KUKA KRL program: EPS_2_25748_MH02A_A_20260121065856.src

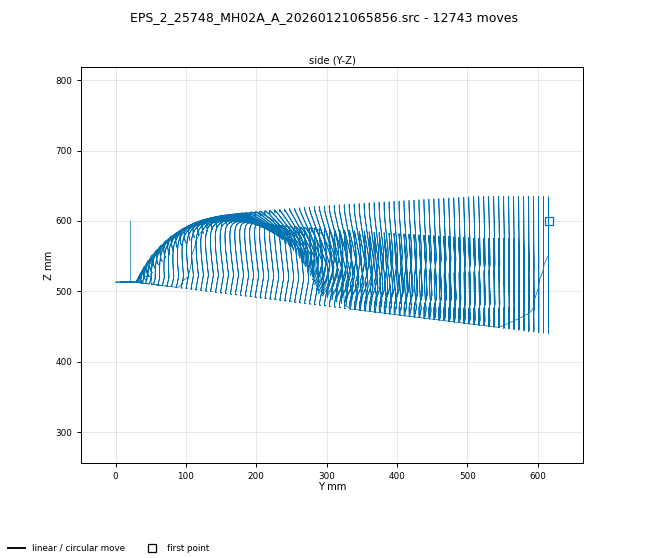
[picture p0: tool path of EPS_2_25748_MH02A_A_20260121065856.src, 12743 of 12745 moves have a stored position in this frame; points joined in program order, loops and branches not executed]
&ACCESS RVP
&REL 4
&COMMENT QRS 19112012
&PARAM EDITMASK = *
DEF PART()
EXT BAS (BAS_COMMAND :IN,REAL :IN )
INT I
BAS (#INITMOV,0 )

;KUKA QRS Post kuka4.cps  Date:22-06-2017 !

File_ID=2997

QRS_PRE_INIT()

;Init var - Until changes are made in qrs_pre_init
Outlet_Square_prg=0
Inlet_1_Square_prg=0
Inlet_2_Square_prg=0
Inlet_3_Square_prg=0
Inlet_4_Square_prg=0
Inlet_5_Square_prg=0

Outlet_1={X 0.000, Y 515.340, Z 534.500, B 0.000, E1 0.000 }
Inlet_1={X 0.000, Y 519.690, Z 474.500, B 0.000, E1 90.000 }
Inlet_2={X 0.000, Y 519.690, Z 474.500, B 0.000, E1 270.000 }
Outlet_1_type=201
Inlet_1_type=201
Inlet_2_type=201
;QRS#1=Sidecore dimensions
;QRS#2=200-8" PVC SDR 35
;QRS#3=200-8" PVC SDR 35
;QRS#4=200-8" PVC SDR 35
;QRS#5=
;QRS#6=
;QRS#7=
;QRS#8=
;QRS#9=12-08 PSX
;QRS#10=12-08 PSX
;QRS#11=12-08 PSX
;QRS#12=
;QRS#13=
;QRS#14=
;QRS#15=
;QRS#16=1220x127x914 3'
;QRS#17=EPS Height
;QRS#18=635
;QRS#19=*
;QRS#20= UPDATED VERSION 22-06-2017
;QRS#21=*
Outlet_Square=0100
Inlet_1_Square=0100
Inlet_2_Square=0100
Inlet_3_Square=0
Inlet_4_Square=0
Inlet_5_Square=0
Mill_Square=1
Outlet_Square_Prg=204
Inlet_1_Square_prg=204
Inlet_2_Square_prg=204

QRS_INIT()

$ADVANCE=5

; T1
PTP {E1 173.497,E2 173.497}
PTP {X 0,Y 615.499,A -85,B 0,C 180,E1 173.497,E2 173.497,E3 0,E4 0,E5 0,E6 0}
QRS_SPEED_INIT()
LIN {X 0,Y 615.499,Z 600,A -85,B 0,C 180,E1 173.497,E2 173.497,E3 0,E4 0,E5 0,E6 0} C_VEL
LIN {X 0,Y 615.499,Z 565.725,A -85,B 0,C 180,E1 173.497,E2 173.497} C_VEL
LIN {X 0,Y 615.499,Z 554.844,A -85,B 0,C 180,E1 173.497,E2 173.497} C_VEL
LIN {X 0,Y 615.497,Z 553.2,A -85,B 0,C 180,E1 173.417,E2 173.417} C_VEL
LIN {X 0,Y 615.497,Z 545.535,A -85,B 0,C 180,E1 172.454,E2 172.454} C_VEL
LIN {X 0,Y 615.498,Z 535.756,A -85,B 0,C 180,E1 171.463,E2 171.463} C_VEL
LIN {X 0,Y 615.498,Z 525.49,A -85,B 0,C 180,E1 170.635,E2 170.635} C_VEL
LIN {X 0,Y 615.481,Z 513.928,A -85,B 0,C 180,E1 169.888,E2 169.888} C_VEL
LIN {X 0,Y 615.482,Z 502.142,A -85,B 0,C 180,E1 169.296,E2 169.296} C_VEL
LIN {X 0,Y 615.483,Z 489.153,A -85,B 0,C 180,E1 168.807,E2 168.807} C_VEL
LIN {X 0,Y 615.487,Z 476.549,A -85,B 0,C 180,E1 168.473,E2 168.473} C_VEL
LIN {X 0,Y 615.484,Z 471.197,A -85,B 0,C 180,E1 168.369,E2 168.369} C_VEL
LIN {X 0,Y 615.476,Z 467.928,A -85,B 0,C 180,E1 166.073,E2 166.073} C_VEL
LIN {X 0,Y 615.492,Z 464.179,A -85,B 0,C 180,E1 163.413,E2 163.413} C_VEL
LIN {X 0,Y 615.485,Z 460.37,A -85,B 0,C 180,E1 160.662,E2 160.662} C_VEL
LIN {X 0,Y 615.48,Z 456.547,A -85,B 0,C 180,E1 157.863,E2 157.863} C_VEL
LIN {X 0,Y 615.476,Z 452.731,A -85,B 0,C 180,E1 155.007,E2 155.007} C_VEL
LIN {X 0,Y 615.481,Z 449.861,A -85,B 0,C 180,E1 152.822,E2 152.822} C_VEL
LIN {X 0,Y 615.498,Z 446.504,A -85,B 0,C 180,E1 150.204,E2 150.204} C_VEL
LIN {X 0,Y 615.485,Z 443.191,A -85,B 0,C 180,E1 147.542,E2 147.542} C_VEL
LIN {X 0,Y 615.48,Z 440.363,A -85,B 0,C 180,E1 145.184,E2 145.184} C_VEL
LIN {X 0,Y 615.477,Z 439.691,A -85,B 0,C 180,E1 144.168,E2 144.168} C_VEL
LIN {X 0,Y 615.484,Z 439.689,A -85,B 0,C 180,E1 141.931,E2 141.931} C_VEL
LIN {X 0,Y 615.479,Z 439.698,A -85,B 0,C 180,E1 139.392,E2 139.392} C_VEL
LIN {X 0,Y 615.497,Z 439.687,A -85,B 0,C 180,E1 136.756,E2 136.756} C_VEL
LIN {X 0,Y 615.49,Z 439.69,A -85,B 0,C 180,E1 133.997,E2 133.997} C_VEL
LIN {X 0,Y 615.491,Z 439.7,A -85,B 0,C 180,E1 131.094,E2 131.094} C_VEL
LIN {X 0,Y 615.486,Z 439.692,A -85,B 0,C 180,E1 128.905,E2 128.905} C_VEL
LIN {X 0,Y 615.479,Z 439.691,A -85,B 0,C 180,E1 126.426,E2 126.426} C_VEL
LIN {X 0,Y 615.496,Z 439.697,A -85,B 0,C 180,E1 124.022,E2 124.022} C_VEL
LIN {X 0,Y 615.487,Z 439.688,A -85,B 0,C 180,E1 121.686,E2 121.686} C_VEL
LIN {X 0,Y 615.484,Z 439.693,A -85,B 0,C 180,E1 119.407,E2 119.407} C_VEL
LIN {X 0,Y 615.486,Z 439.696,A -85,B 0,C 180,E1 117.044,E2 117.044} C_VEL
LIN {X 0,Y 615.477,Z 439.694,A -85,B 0,C 180,E1 114.273,E2 114.273} C_VEL
LIN {X 0,Y 615.477,Z 439.69,A -85,B 0,C 180,E1 111.432,E2 111.432} C_VEL
LIN {X 0,Y 615.491,Z 439.699,A -85,B 0,C 180,E1 108.604,E2 108.604} C_VEL
LIN {X 0,Y 615.489,Z 439.688,A -85,B 0,C 180,E1 105.905,E2 105.905} C_VEL
LIN {X 0,Y 615.482,Z 439.694,A -85,B 0,C 180,E1 103.201,E2 103.201} C_VEL
LIN {X 0,Y 615.478,Z 439.694,A -85,B 0,C 180,E1 100.527,E2 100.527} C_VEL
LIN {X 0,Y 615.489,Z 439.689,A -85,B 0,C 180,E1 97.876,E2 97.876} C_VEL
LIN {X 0,Y 615.482,Z 439.696,A -85,B 0,C 180,E1 95.241,E2 95.241} C_VEL
LIN {X 0,Y 615.477,Z 439.691,A -85,B 0,C 180,E1 92.618,E2 92.618} C_VEL
LIN {X 0,Y 615.492,Z 439.696,A -85,B 0,C 180,E1 90,E2 90} C_VEL
LIN {X 0,Y 615.478,Z 439.69,A -85,B 0,C 180,E1 87.382,E2 87.382} C_VEL
LIN {X 0,Y 615.494,Z 439.698,A -85,B 0,C 180,E1 84.759,E2 84.759} C_VEL
LIN {X 0,Y 615.487,Z 439.688,A -85,B 0,C 180,E1 82.124,E2 82.124} C_VEL
LIN {X 0,Y 615.494,Z 439.7,A -85,B 0,C 180,E1 79.473,E2 79.473} C_VEL
LIN {X 0,Y 615.482,Z 439.689,A -85,B 0,C 180,E1 76.799,E2 76.799} C_VEL
LIN {X 0,Y 615.491,Z 439.694,A -85,B 0,C 180,E1 74.095,E2 74.095} C_VEL
LIN {X 0,Y 615.483,Z 439.693,A -85,B 0,C 180,E1 71.354,E2 71.354} C_VEL
LIN {X 0,Y 615.477,Z 439.691,A -85,B 0,C 180,E1 68.568,E2 68.568} C_VEL
LIN {X 0,Y 615.485,Z 439.701,A -85,B 0,C 180,E1 65.728,E2 65.728} C_VEL
LIN {X 0,Y 615.486,Z 439.689,A -85,B 0,C 180,E1 62.956,E2 62.956} C_VEL
LIN {X 0,Y 615.498,Z 439.689,A -85,B 0,C 180,E1 60.205,E2 60.205} C_VEL
LIN {X 0,Y 615.48,Z 439.695,A -85,B 0,C 180,E1 57.542,E2 57.542} C_VEL
LIN {X 0,Y 615.499,Z 439.691,A -85,B 0,C 180,E1 55.185,E2 55.185} C_VEL
LIN {X 0,Y 615.477,Z 439.69,A -85,B 0,C 180,E1 52.757,E2 52.757} C_VEL
LIN {X 0,Y 615.477,Z 439.694,A -85,B 0,C 180,E1 49.913,E2 49.913} C_VEL
LIN {X 0,Y 615.475,Z 439.69,A -85,B 0,C 180,E1 47.646,E2 47.646} C_VEL
LIN {X 0,Y 615.483,Z 439.696,A -85,B 0,C 180,E1 44.931,E2 44.931} C_VEL
LIN {X 0,Y 615.494,Z 439.692,A -85,B 0,C 180,E1 42.08,E2 42.08} C_VEL
LIN {X 0,Y 615.478,Z 439.696,A -85,B 0,C 180,E1 39.751,E2 39.751} C_VEL
LIN {X 0,Y 615.485,Z 439.694,A -85,B 0,C 180,E1 36.936,E2 36.936} C_VEL
LIN {X 0,Y 615.48,Z 439.689,A -85,B 0,C 180,E1 35.617,E2 35.617} C_VEL
LIN {X 0,Y 615.493,Z 440.123,A -85,B 0,C 180,E1 34.701,E2 34.701} C_VEL
LIN {X 0,Y 615.495,Z 443.189,A -85,B 0,C 180,E1 32.331,E2 32.331} C_VEL
LIN {X 0,Y 615.487,Z 446.882,A -85,B 0,C 180,E1 29.407,E2 29.407} C_VEL
LIN {X 0,Y 615.48,Z 449.92,A -85,B 0,C 180,E1 27.043,E2 27.043} C_VEL
LIN {X 0,Y 615.492,Z 453.568,A -85,B 0,C 180,E1 24.272,E2 24.272} C_VEL
LIN {X 0,Y 615.494,Z 457.377,A -85,B 0,C 180,E1 21.432,E2 21.432} C_VEL
LIN {X 0,Y 615.494,Z 461.252,A -85,B 0,C 180,E1 18.606,E2 18.606} C_VEL
LIN {X 0,Y 615.476,Z 465.011,A -85,B 0,C 180,E1 15.906,E2 15.906} C_VEL
LIN {X 0,Y 615.493,Z 468.827,A -85,B 0,C 180,E1 13.201,E2 13.201} C_VEL
LIN {X 0,Y 615.484,Z 471.187,A -85,B 0,C 180,E1 11.548,E2 11.548} C_VEL
LIN {X 0,Y 615.485,Z 486.247,A -85,B 0,C 180,E1 11.193,E2 11.193} C_VEL
LIN {X 0,Y 615.48,Z 497.908,A -85,B 0,C 180,E1 10.793,E2 10.793} C_VEL
LIN {X 0,Y 615.486,Z 509.192,A -85,B 0,C 180,E1 10.278,E2 10.278} C_VEL
LIN {X 0,Y 615.492,Z 520.573,A -85,B 0,C 180,E1 9.613,E2 9.613} C_VEL
LIN {X 0,Y 615.498,Z 530.82,A -85,B 0,C 180,E1 8.868,E2 8.868} C_VEL
LIN {X 0,Y 615.498,Z 540.032,A -85,B 0,C 180,E1 8.041,E2 8.041} C_VEL
LIN {X 0,Y 615.499,Z 548.89,A -85,B 0,C 180,E1 7.058,E2 7.058} C_VEL
LIN {X 0,Y 615.497,Z 556.122,A -85,B 0,C 180,E1 6.063,E2 6.063} C_VEL
LIN {X 0,Y 615.497,Z 560.957,A -85,B 0,C 180,E1 5.241,E2 5.241} C_VEL
LIN {X 0,Y 615.493,Z 565.657,A -85,B 0,C 180,E1 4.257,E2 4.257} C_VEL
LIN {X 0,Y 615.495,Z 569.254,A -85,B 0,C 180,E1 3.273,E2 3.273} C_VEL
LIN {X 0,Y 615.496,Z 571.114,A -85,B 0,C 180,E1 2.618,E2 2.618} C_VEL
LIN {X 0,Y 615.497,Z 572.533,A -85,B 0,C 180,E1 1.963,E2 1.963} C_VEL
LIN {X 0,Y 615.497,Z 574.141,A -85,B 0,C 180,E1 0.654,E2 0.654} C_VEL
LIN {X 0,Y 615.494,Z 574.384,A -85,B 0,C 180,E1 0,E2 0} C_VEL
LIN {X 0,Y 615.495,Z 574.206,A -85,B 0,C 180,E1 -0.654,E2 -0.654} C_VEL
LIN {X 0,Y 615.496,Z 572.683,A -85,B 0,C 180,E1 -1.963,E2 -1.963} C_VEL
LIN {X 0,Y 615.498,Z 571.341,A -85,B 0,C 180,E1 -2.618,E2 -2.618} C_VEL
LIN {X 0,Y 615.498,Z 568.494,A -85,B 0,C 180,E1 -3.6,E2 -3.6} C_VEL
LIN {X 0,Y 615.498,Z 564.635,A -85,B 0,C 180,E1 -4.584,E2 -4.584} C_VEL
LIN {X 0,Y 615.499,Z 559.652,A -85,B 0,C 180,E1 -5.57,E2 -5.57} C_VEL
LIN {X 0,Y 615.496,Z 553.208,A -85,B 0,C 180,E1 -6.582,E2 -6.582} C_VEL
LIN {X 0,Y 615.497,Z 545.538,A -85,B 0,C 180,E1 -7.545,E2 -7.545} C_VEL
LIN {X 0,Y 615.498,Z 535.76,A -85,B 0,C 180,E1 -8.536,E2 -8.536} C_VEL
LIN {X 0,Y 615.498,Z 525.494,A -85,B 0,C 180,E1 -9.364,E2 -9.364} C_VEL
LIN {X 0,Y 615.479,Z 513.933,A -85,B 0,C 180,E1 -10.111,E2 -10.111} C_VEL
LIN {X 0,Y 615.482,Z 502.146,A -85,B 0,C 180,E1 -10.704,E2 -10.704} C_VEL
LIN {X 0,Y 615.483,Z 489.163,A -85,B 0,C 180,E1 -11.193,E2 -11.193} C_VEL
LIN {X 0,Y 615.487,Z 476.563,A -85,B 0,C 180,E1 -11.527,E2 -11.527} C_VEL
LIN {X 0,Y 615.484,Z 471.197,A -85,B 0,C 180,E1 -11.631,E2 -11.631} C_VEL
LIN {X 0,Y 615.476,Z 467.929,A -85,B 0,C 180,E1 -13.927,E2 -13.927} C_VEL
LIN {X 0,Y 615.487,Z 464.181,A -85,B 0,C 180,E1 -16.587,E2 -16.587} C_VEL
LIN {X 0,Y 615.489,Z 460.369,A -85,B 0,C 180,E1 -19.338,E2 -19.338} C_VEL
LIN {X 0,Y 615.479,Z 456.548,A -85,B 0,C 180,E1 -22.137,E2 -22.137} C_VEL
LIN {X 0,Y 615.491,Z 453.686,A -85,B 0,C 180,E1 -24.272,E2 -24.272} C_VEL
LIN {X 0,Y 615.481,Z 449.862,A -85,B 0,C 180,E1 -27.177,E2 -27.177} C_VEL
LIN {X 0,Y 615.497,Z 446.505,A -85,B 0,C 180,E1 -29.796,E2 -29.796} C_VEL
LIN {X 0,Y 615.493,Z 443.035,A -85,B 0,C 180,E1 -32.457,E2 -32.457} C_VEL
LIN {X 0,Y 615.484,Z 439.698,A -85,B 0,C 180,E1 -34.7,E2 -34.7} C_VEL
LIN {X 0,Y 615.491,Z 439.696,A -85,B 0,C 180,E1 -37.242,E2 -37.242} C_VEL
LIN {X 0,Y 615.486,Z 439.695,A -85,B 0,C 180,E1 -40.089,E2 -40.089} C_VEL
LIN {X 0,Y 615.493,Z 439.696,A -85,B 0,C 180,E1 -42.353,E2 -42.353} C_VEL
LIN {X 0,Y 615.488,Z 439.695,A -85,B 0,C 180,E1 -45.069,E2 -45.069} C_VEL
LIN {X 0,Y 615.48,Z 439.696,A -85,B 0,C 180,E1 -47.921,E2 -47.921} C_VEL
LIN {X 0,Y 615.494,Z 439.693,A -85,B 0,C 180,E1 -50.25,E2 -50.25} C_VEL
LIN {X 0,Y 615.482,Z 439.696,A -85,B 0,C 180,E1 -53.064,E2 -53.064} C_VEL
LIN {X 0,Y 615.487,Z 439.699,A -85,B 0,C 180,E1 -54.484,E2 -54.484} C_VEL
LIN {X 0,Y 615.488,Z 448.578,A -85,B 0,C 180,E1 -57.154,E2 -57.154} C_VEL
LIN {X 0,Y 615.48,Z 457.828,A -85,B 0,C 180,E1 -59.839,E2 -59.839} C_VEL
LIN {X 0,Y 615.481,Z 467.078,A -85,B 0,C 180,E1 -62.454,E2 -62.454} C_VEL
LIN {X 0,Y 615.488,Z 476.316,A -85,B 0,C 180,E1 -65.008,E2 -65.008} C_VEL
LIN {X 0,Y 615.482,Z 486.871,A -85,B 0,C 180,E1 -67.863,E2 -67.863} C_VEL
LIN {X 0,Y 615.475,Z 497.419,A -85,B 0,C 180,E1 -70.662,E2 -70.662} C_VEL
LIN {X 0,Y 615.48,Z 507.958,A -85,B 0,C 180,E1 -73.413,E2 -73.413} C_VEL
LIN {X 0,Y 615.493,Z 518.495,A -85,B 0,C 180,E1 -76.126,E2 -76.126} C_VEL
LIN {X 0,Y 615.487,Z 527.208,A -85,B 0,C 180,E1 -78.348,E2 -78.348} C_VEL
LIN {X 0,Y 615.496,Z 541.819,A -85,B 0,C 180,E1 -78.64,E2 -78.64} C_VEL
LIN {X 0,Y 615.49,Z 554.558,A -85,B 0,C 180,E1 -79.036,E2 -79.036} C_VEL
LIN {X 0,Y 615.477,Z 566.767,A -85,B 0,C 180,E1 -79.556,E2 -79.556} C_VEL
LIN {X 0,Y 615.491,Z 577.387,A -85,B 0,C 180,E1 -80.138,E2 -80.138} C_VEL
LIN {X 0,Y 615.498,Z 588.231,A -85,B 0,C 180,E1 -80.884,E2 -80.884} C_VEL
LIN {X 0,Y 615.497,Z 598.811,A -85,B 0,C 180,E1 -81.794,E2 -81.794} C_VEL
LIN {X 0,Y 615.498,Z 606.606,A -85,B 0,C 180,E1 -82.62,E2 -82.62} C_VEL
LIN {X 0,Y 615.496,Z 614.203,A -85,B 0,C 180,E1 -83.608,E2 -83.608} C_VEL
LIN {X 0,Y 615.498,Z 621.204,A -85,B 0,C 180,E1 -84.759,E2 -84.759} C_VEL
LIN {X 0,Y 615.493,Z 625.851,A -85,B 0,C 180,E1 -85.744,E2 -85.744} C_VEL
LIN {X 0,Y 615.495,Z 629.398,A -85,B 0,C 180,E1 -86.727,E2 -86.727} C_VEL
LIN {X 0,Y 615.497,Z 631.233,A -85,B 0,C 180,E1 -87.382,E2 -87.382} C_VEL
LIN {X 0,Y 615.497,Z 632.608,A -85,B 0,C 180,E1 -88.037,E2 -88.037} C_VEL
LIN {X 0,Y 615.496,Z 634.174,A -85,B 0,C 180,E1 -89.346,E2 -89.346} C_VEL
LIN {X 0,Y 615.494,Z 634.389,A -85,B 0,C 180,E1 -90,E2 -90} C_VEL
LIN {X 0,Y 615.496,Z 633.58,A -85,B 0,C 180,E1 -91.309,E2 -91.309} C_VEL
LIN {X 0,Y 615.497,Z 632.608,A -85,B 0,C 180,E1 -91.963,E2 -91.963} C_VEL
LIN {X 0,Y 615.497,Z 631.233,A -85,B 0,C 180,E1 -92.618,E2 -92.618} C_VEL
LIN {X 0,Y 615.496,Z 628.349,A -85,B 0,C 180,E1 -93.601,E2 -93.601} C_VEL
LIN {X 0,Y 615.498,Z 624.441,A -85,B 0,C 180,E1 -94.584,E2 -94.584} C_VEL
LIN {X 0,Y 615.499,Z 619.405,A -85,B 0,C 180,E1 -95.57,E2 -95.57} C_VEL
LIN {X 0,Y 615.497,Z 612.869,A -85,B 0,C 180,E1 -96.583,E2 -96.583} C_VEL
LIN {X 0,Y 615.497,Z 605.133,A -85,B 0,C 180,E1 -97.545,E2 -97.545} C_VEL
LIN {X 0,Y 615.498,Z 597.044,A -85,B 0,C 180,E1 -98.371,E2 -98.371} C_VEL
LIN {X 0,Y 615.499,Z 587.167,A -85,B 0,C 180,E1 -99.199,E2 -99.199} C_VEL
LIN {X 0,Y 615.488,Z 575.981,A -85,B 0,C 180,E1 -99.945,E2 -99.945} C_VEL
LIN {X 0,Y 615.478,Z 565.023,A -85,B 0,C 180,E1 -100.527,E2 -100.527} C_VEL
LIN {X 0,Y 615.494,Z 552.485,A -85,B 0,C 180,E1 -101.04,E2 -101.04} C_VEL
LIN {X 0,Y 615.495,Z 540.061,A -85,B 0,C 180,E1 -101.401,E2 -101.401} C_VEL
LIN {X 0,Y 615.487,Z 527.208,A -85,B 0,C 180,E1 -101.652,E2 -101.652} C_VEL
LIN {X 0,Y 615.48,Z 517.063,A -85,B 0,C 180,E1 -104.242,E2 -104.242} C_VEL
LIN {X 0,Y 615.495,Z 506.637,A -85,B 0,C 180,E1 -106.928,E2 -106.928} C_VEL
LIN {X 0,Y 615.485,Z 496.105,A -85,B 0,C 180,E1 -109.685,E2 -109.685} C_VEL
LIN {X 0,Y 615.477,Z 486.101,A -85,B 0,C 180,E1 -112.343,E2 -112.343} C_VEL
LIN {X 0,Y 615.488,Z 476.316,A -85,B 0,C 180,E1 -114.992,E2 -114.992} C_VEL
LIN {X 0,Y 615.481,Z 467.078,A -85,B 0,C 180,E1 -117.546,E2 -117.546} C_VEL
LIN {X 0,Y 615.483,Z 457.828,A -85,B 0,C 180,E1 -120.16,E2 -120.16} C_VEL
LIN {X 0,Y 615.486,Z 448.579,A -85,B 0,C 180,E1 -122.846,E2 -122.846} C_VEL
LIN {X 0,Y 615.485,Z 439.895,A -85,B 0,C 180,E1 -125.516,E2 -125.516} C_VEL
LIN {X 0,Y 615.481,Z 439.698,A -85,B 0,C 180,E1 -128.069,E2 -128.069} C_VEL
LIN {X 0,Y 615.489,Z 439.695,A -85,B 0,C 180,E1 -130.607,E2 -130.607} C_VEL
LIN {X 0,Y 615.476,Z 439.698,A -85,B 0,C 180,E1 -133.246,E2 -133.246} C_VEL
LIN {X 0,Y 615.492,Z 439.698,A -85,B 0,C 180,E1 -136.002,E2 -136.002} C_VEL
LIN {X 0,Y 615.488,Z 439.7,A -85,B 0,C 180,E1 -138.526,E2 -138.526} C_VEL
LIN {X 0,Y 615.496,Z 439.7,A -85,B 0,C 180,E1 -141.096,E2 -141.096} C_VEL
LIN {X 0,Y 615.493,Z 439.7,A -85,B 0,C 180,E1 -143.576,E2 -143.576} C_VEL
LIN {X 0,Y 615.479,Z 439.699,A -85,B 0,C 180,E1 -144.384,E2 -144.384} C_VEL
LIN {X 0,Y 615.497,Z 442.286,A -85,B 0,C 180,E1 -146.764,E2 -146.764} C_VEL
LIN {X 0,Y 615.478,Z 444.973,A -85,B 0,C 180,E1 -149.08,E2 -149.08} C_VEL
LIN {X 0,Y 615.491,Z 448.106,A -85,B 0,C 180,E1 -151.55,E2 -151.55} C_VEL
LIN {X 0,Y 615.49,Z 451.846,A -85,B 0,C 180,E1 -154.431,E2 -154.431} C_VEL
LIN {X 0,Y 615.475,Z 455.48,A -85,B 0,C 180,E1 -157.155,E2 -157.155} C_VEL
LIN {X 0,Y 615.49,Z 458.575,A -85,B 0,C 180,E1 -159.443,E2 -159.443} C_VEL
LIN {X 0,Y 615.477,Z 462.148,A -85,B 0,C 180,E1 -162.043,E2 -162.043} C_VEL
LIN {X 0,Y 615.496,Z 465.971,A -85,B 0,C 180,E1 -164.774,E2 -164.774} C_VEL
LIN {X 0,Y 615.485,Z 469.775,A -85,B 0,C 180,E1 -167.47,E2 -167.47} C_VEL
LIN {X 0,Y 615.486,Z 471.188,A -85,B 0,C 180,E1 -168.452,E2 -168.452} C_VEL
LIN {X 0,Y 615.487,Z 486.259,A -85,B 0,C 180,E1 -168.807,E2 -168.807} C_VEL
LIN {X 0,Y 615.482,Z 498.96,A -85,B 0,C 180,E1 -169.251,E2 -169.251} C_VEL
LIN {X 0,Y 615.482,Z 510.76,A -85,B 0,C 180,E1 -169.806,E2 -169.806} C_VEL
LIN {X 0,Y 615.496,Z 521.849,A -85,B 0,C 180,E1 -170.47,E2 -170.47} C_VEL
LIN {X 0,Y 615.498,Z 530.824,A -85,B 0,C 180,E1 -171.133,E2 -171.133} C_VEL
LIN {X 0,Y 615.498,Z 540.035,A -85,B 0,C 180,E1 -171.959,E2 -171.959} C_VEL
LIN {X 0,Y 615.499,Z 548.893,A -85,B 0,C 180,E1 -172.943,E2 -172.943} C_VEL
LIN {X 0,Y 615.497,Z 556.124,A -85,B 0,C 180,E1 -173.937,E2 -173.937} C_VEL
LIN {X 0,Y 615.498,Z 560.959,A -85,B 0,C 180,E1 -174.759,E2 -174.759} C_VEL
LIN {X 0,Y 615.493,Z 565.658,A -85,B 0,C 180,E1 -175.744,E2 -175.744} C_VEL
LIN {X 0,Y 615.496,Z 569.255,A -85,B 0,C 180,E1 -176.727,E2 -176.727} C_VEL
LIN {X 0,Y 615.496,Z 571.115,A -85,B 0,C 180,E1 -177.382,E2 -177.382} C_VEL
LIN {X 0,Y 615.497,Z 572.534,A -85,B 0,C 180,E1 -178.037,E2 -178.037} C_VEL
LIN {X 0,Y 615.496,Z 574.142,A -85,B 0,C 180,E1 -179.346,E2 -179.346} C_VEL
LIN {X 0,Y 615.494,Z 574.384,A -85,B 0,C 180,E1 -180,E2 -180} C_VEL
LIN {X 0,Y 615.496,Z 574.205,A -85,B 0,C 180,E1 -180.654,E2 -180.654} C_VEL
LIN {X 0,Y 615.496,Z 572.683,A -85,B 0,C 180,E1 -181.963,E2 -181.963} C_VEL
LIN {X 0,Y 615.498,Z 571.341,A -85,B 0,C 180,E1 -182.618,E2 -182.618} C_VEL
LIN {X 0,Y 615.497,Z 568.493,A -85,B 0,C 180,E1 -183.601,E2 -183.601} C_VEL
LIN {X 0,Y 615.499,Z 564.633,A -85,B 0,C 180,E1 -184.585,E2 -184.585} C_VEL
LIN {X 0,Y 615.498,Z 559.65,A -85,B 0,C 180,E1 -185.57,E2 -185.57} C_VEL
LIN {X 0,Y 615.497,Z 553.2,A -85,B 0,C 180,E1 -186.583,E2 -186.583} C_VEL
LIN {X 0,Y 614.829,Z 550.018,A -85,B 0,C 180,E1 -187.032,E2 -187.032} C_VEL
LIN {X 0,Y 611.988,Z 544.445,A -85,B 0,C 180,E1 -187.749,E2 -187.749} C_VEL
LIN {X 0,Y 609.138,Z 538.168,A -85,B 0,C 180,E1 -188.43,E2 -188.43} C_VEL
LIN {X 0,Y 608.477,Z 533.927,A -85,B 0,C 180,E1 -188.82,E2 -188.82} C_VEL
LIN {X 0,Y 608.494,Z 523.387,A -85,B 0,C 180,E1 -189.641,E2 -189.641} C_VEL
LIN {X 0,Y 608.49,Z 512.607,A -85,B 0,C 180,E1 -190.313,E2 -190.313} C_VEL
LIN {X 0,Y 608.507,Z 500.307,A -85,B 0,C 180,E1 -190.913,E2 -190.913} C_VEL
LIN {X 0,Y 608.522,Z 487.959,A -85,B 0,C 180,E1 -191.365,E2 -191.365} C_VEL
LIN {X 0,Y 608.545,Z 475.645,A -85,B 0,C 180,E1 -191.681,E2 -191.681} C_VEL
LIN {X 0,Y 608.429,Z 471.674,A -85,B 0,C 180,E1 -191.768,E2 -191.768} C_VEL
LIN {X 0,Y 608.43,Z 468.46,A -85,B 0,C 180,E1 -194.039,E2 -194.039} C_VEL
LIN {X 0,Y 608.421,Z 464.614,A -85,B 0,C 180,E1 -196.785,E2 -196.785} C_VEL
LIN {X 0,Y 608.41,Z 460.769,A -85,B 0,C 180,E1 -199.572,E2 -199.572} C_VEL
LIN {X 0,Y 608.437,Z 456.924,A -85,B 0,C 180,E1 -202.407,E2 -202.407} C_VEL
LIN {X 0,Y 608.425,Z 453.078,A -85,B 0,C 180,E1 -205.302,E2 -205.302} C_VEL
LIN {X 0,Y 608.435,Z 449.232,A -85,B 0,C 180,E1 -208.268,E2 -208.268} C_VEL
LIN {X 0,Y 608.431,Z 446.348,A -85,B 0,C 180,E1 -210.547,E2 -210.547} C_VEL
LIN {X 0,Y 608.431,Z 443.522,A -85,B 0,C 180,E1 -212.882,E2 -212.882} C_VEL
LIN {X 0,Y 608.41,Z 440.703,A -85,B 0,C 180,E1 -215.28,E2 -215.28} C_VEL
LIN {X 0,Y 608.468,Z 440.688,A -85,B 0,C 180,E1 -217.747,E2 -217.747} C_VEL
LIN {X 0,Y 608.448,Z 440.698,A -85,B 0,C 180,E1 -220.328,E2 -220.328} C_VEL
LIN {X 0,Y 608.452,Z 440.69,A -85,B 0,C 180,E1 -222.96,E2 -222.96} C_VEL
LIN {X 0,Y 608.458,Z 440.695,A -85,B 0,C 180,E1 -225.737,E2 -225.737} C_VEL
LIN {X 0,Y 608.464,Z 440.692,A -85,B 0,C 180,E1 -228.658,E2 -228.658} C_VEL
LIN {X 0,Y 608.441,Z 440.692,A -85,B 0,C 180,E1 -231.41,E2 -231.41} C_VEL
LIN {X 0,Y 608.452,Z 440.695,A -85,B 0,C 180,E1 -233.955,E2 -233.955} C_VEL
LIN {X 0,Y 608.453,Z 440.692,A -85,B 0,C 180,E1 -236.328,E2 -236.328} C_VEL
LIN {X 0,Y 608.45,Z 440.691,A -85,B 0,C 180,E1 -238.733,E2 -238.733} C_VEL
LIN {X 0,Y 608.47,Z 440.69,A -85,B 0,C 180,E1 -241.382,E2 -241.382} C_VEL
LIN {X 0,Y 608.483,Z 440.692,A -85,B 0,C 180,E1 -244.278,E2 -244.278} C_VEL
LIN {X 0,Y 608.45,Z 440.69,A -85,B 0,C 180,E1 -246.876,E2 -246.876} C_VEL
LIN {X 0,Y 608.468,Z 440.694,A -85,B 0,C 180,E1 -249.726,E2 -249.726} C_VEL
LIN {X 0,Y 608.453,Z 440.692,A -85,B 0,C 180,E1 -252.523,E2 -252.523} C_VEL
LIN {X 0,Y 608.471,Z 440.689,A -85,B 0,C 180,E1 -255.279,E2 -255.279} C_VEL
LIN {X 0,Y 608.462,Z 440.694,A -85,B 0,C 180,E1 -258,E2 -258} C_VEL
LIN {X 0,Y 608.467,Z 440.688,A -85,B 0,C 180,E1 -260.694,E2 -260.694} C_VEL
LIN {X 0,Y 608.465,Z 440.696,A -85,B 0,C 180,E1 -263.384,E2 -263.384} C_VEL
LIN {X 0,Y 608.457,Z 440.69,A -85,B 0,C 180,E1 -266.026,E2 -266.026} C_VEL
LIN {X 0,Y 608.466,Z 440.693,A -85,B 0,C 180,E1 -268.676,E2 -268.676} C_VEL
LIN {X 0,Y 608.466,Z 440.689,A -85,B 0,C 180,E1 -271.324,E2 -271.324} C_VEL
LIN {X 0,Y 608.46,Z 440.692,A -85,B 0,C 180,E1 -273.974,E2 -273.974} C_VEL
LIN {X 0,Y 608.447,Z 440.693,A -85,B 0,C 180,E1 -276.633,E2 -276.633} C_VEL
LIN {X 0,Y 608.467,Z 440.689,A -85,B 0,C 180,E1 -279.306,E2 -279.306} C_VEL
LIN {X 0,Y 608.463,Z 440.694,A -85,B 0,C 180,E1 -282,E2 -282} C_VEL
LIN {X 0,Y 608.47,Z 440.688,A -85,B 0,C 180,E1 -284.721,E2 -284.721} C_VEL
LIN {X 0,Y 608.46,Z 440.695,A -85,B 0,C 180,E1 -287.476,E2 -287.476} C_VEL
LIN {X 0,Y 608.463,Z 440.69,A -85,B 0,C 180,E1 -290.274,E2 -290.274} C_VEL
LIN {X 0,Y 608.45,Z 440.691,A -85,B 0,C 180,E1 -293.124,E2 -293.124} C_VEL
LIN {X 0,Y 608.472,Z 440.692,A -85,B 0,C 180,E1 -295.72,E2 -295.72} C_VEL
LIN {X 0,Y 608.446,Z 440.691,A -85,B 0,C 180,E1 -298.267,E2 -298.267} C_VEL
LIN {X 0,Y 608.453,Z 440.691,A -85,B 0,C 180,E1 -300.546,E2 -300.546} C_VEL
LIN {X 0,Y 608.453,Z 440.697,A -85,B 0,C 180,E1 -302.88,E2 -302.88} C_VEL
LIN {X 0,Y 608.447,Z 440.691,A -85,B 0,C 180,E1 -305.278,E2 -305.278} C_VEL
LIN {X 0,Y 608.467,Z 440.693,A -85,B 0,C 180,E1 -307.747,E2 -307.747} C_VEL
LIN {X 0,Y 608.445,Z 440.691,A -85,B 0,C 180,E1 -310.327,E2 -310.327} C_VEL
LIN {X 0,Y 608.48,Z 440.691,A -85,B 0,C 180,E1 -313.309,E2 -313.309} C_VEL
LIN {X 0,Y 608.474,Z 440.69,A -85,B 0,C 180,E1 -316.13,E2 -316.13} C_VEL
LIN {X 0,Y 608.452,Z 440.691,A -85,B 0,C 180,E1 -318.823,E2 -318.823} C_VEL
LIN {X 0,Y 608.466,Z 440.695,A -85,B 0,C 180,E1 -321.76,E2 -321.76} C_VEL
LIN {X 0,Y 608.449,Z 440.691,A -85,B 0,C 180,E1 -323.955,E2 -323.955} C_VEL
LIN {X 0,Y 608.429,Z 440.701,A -85,B 0,C 180,E1 -325.098,E2 -325.098} C_VEL
LIN {X 0,Y 608.434,Z 443.739,A -85,B 0,C 180,E1 -327.482,E2 -327.482} C_VEL
LIN {X 0,Y 608.444,Z 447.196,A -85,B 0,C 180,E1 -330.219,E2 -330.219} C_VEL
LIN {X 0,Y 608.427,Z 450.493,A -85,B 0,C 180,E1 -332.803,E2 -332.803} C_VEL
LIN {X 0,Y 608.423,Z 453.921,A -85,B 0,C 180,E1 -335.427,E2 -335.427} C_VEL
LIN {X 0,Y 608.418,Z 457.764,A -85,B 0,C 180,E1 -338.306,E2 -338.306} C_VEL
LIN {X 0,Y 608.425,Z 461.607,A -85,B 0,C 180,E1 -341.129,E2 -341.129} C_VEL
LIN {X 0,Y 608.421,Z 465.45,A -85,B 0,C 180,E1 -343.905,E2 -343.905} C_VEL
LIN {X 0,Y 608.432,Z 469.294,A -85,B 0,C 180,E1 -346.643,E2 -346.643} C_VEL
LIN {X 0,Y 608.429,Z 471.666,A -85,B 0,C 180,E1 -348.316,E2 -348.316} C_VEL
LIN {X 0,Y 608.53,Z 487.596,A -85,B 0,C 180,E1 -348.713,E2 -348.713} C_VEL
LIN {X 0,Y 608.503,Z 500.161,A -85,B 0,C 180,E1 -349.171,E2 -349.171} C_VEL
LIN {X 0,Y 608.481,Z 512.498,A -85,B 0,C 180,E1 -349.771,E2 -349.771} C_VEL
LIN {X 0,Y 608.488,Z 523.298,A -85,B 0,C 180,E1 -350.443,E2 -350.443} C_VEL
LIN {X 0,Y 608.477,Z 533.071,A -85,B 0,C 180,E1 -351.197,E2 -351.197} C_VEL
LIN {X 0,Y 608.46,Z 541.971,A -85,B 0,C 180,E1 -352.033,E2 -352.033} C_VEL
LIN {X 0,Y 608.465,Z 550.661,A -85,B 0,C 180,E1 -353.034,E2 -353.034} C_VEL
LIN {X 0,Y 608.439,Z 557.591,A -85,B 0,C 180,E1 -354.033,E2 -354.033} C_VEL
LIN {X 0,Y 608.436,Z 563.145,A -85,B 0,C 180,E1 -355.03,E2 -355.03} C_VEL
LIN {X 0,Y 608.434,Z 567.506,A -85,B 0,C 180,E1 -356.026,E2 -356.026} C_VEL
LIN {X 0,Y 608.426,Z 569.812,A -85,B 0,C 180,E1 -356.689,E2 -356.689} C_VEL
LIN {X 0,Y 608.425,Z 571.689,A -85,B 0,C 180,E1 -357.352,E2 -357.352} C_VEL
LIN {X 0,Y 608.442,Z 573.126,A -85,B 0,C 180,E1 -358.014,E2 -358.014} C_VEL
LIN {X 0,Y 608.44,Z 574.752,A -85,B 0,C 180,E1 -359.338,E2 -359.338} C_VEL
LIN {X 0,Y 608.434,Z 574.995,A -85,B 0,C 180,E1 -360,E2 -360} C_VEL
LIN {X 0,Y 608.438,Z 574.815,A -85,B 0,C 180,E1 -360.662,E2 -360.662} C_VEL
LIN {X 0,Y 608.441,Z 573.276,A -85,B 0,C 180,E1 -361.986,E2 -361.986} C_VEL
LIN {X 0,Y 608.426,Z 571.919,A -85,B 0,C 180,E1 -362.648,E2 -362.648} C_VEL
LIN {X 0,Y 608.451,Z 569.043,A -85,B 0,C 180,E1 -363.642,E2 -363.642} C_VEL
LIN {X 0,Y 608.433,Z 565.144,A -85,B 0,C 180,E1 -364.638,E2 -364.638} C_VEL
LIN {X 0,Y 608.45,Z 560.113,A -85,B 0,C 180,E1 -365.634,E2 -365.634} C_VEL
LIN {X 0,Y 608.441,Z 553.793,A -85,B 0,C 180,E1 -366.633,E2 -366.633} C_VEL
LIN {X 0,Y 608.475,Z 545.881,A -85,B 0,C 180,E1 -367.633,E2 -367.633} C_VEL
LIN {X 0,Y 608.472,Z 536.037,A -85,B 0,C 180,E1 -368.636,E2 -368.636} C_VEL
LIN {X 0,Y 608.48,Z 525.711,A -85,B 0,C 180,E1 -369.473,E2 -369.473} C_VEL
LIN {X 0,Y 608.477,Z 514.099,A -85,B 0,C 180,E1 -370.229,E2 -370.229} C_VEL
LIN {X 0,Y 608.502,Z 502.086,A -85,B 0,C 180,E1 -370.836,E2 -370.836} C_VEL
LIN {X 0,Y 608.529,Z 489.255,A -85,B 0,C 180,E1 -371.323,E2 -371.323} C_VEL
LIN {X 0,Y 608.535,Z 476.633,A -85,B 0,C 180,E1 -371.66,E2 -371.66} C_VEL
LIN {X 0,Y 608.429,Z 471.674,A -85,B 0,C 180,E1 -371.768,E2 -371.768} C_VEL
LIN {X 0,Y 608.42,Z 468.46,A -85,B 0,C 180,E1 -374.039,E2 -374.039} C_VEL
LIN {X 0,Y 608.419,Z 464.615,A -85,B 0,C 180,E1 -376.785,E2 -376.785} C_VEL
LIN {X 0,Y 608.412,Z 460.77,A -85,B 0,C 180,E1 -379.572,E2 -379.572} C_VEL
LIN {X 0,Y 608.432,Z 456.84,A -85,B 0,C 180,E1 -382.469,E2 -382.469} C_VEL
LIN {X 0,Y 608.427,Z 453.078,A -85,B 0,C 180,E1 -385.302,E2 -385.302} C_VEL
LIN {X 0,Y 608.435,Z 449.233,A -85,B 0,C 180,E1 -388.268,E2 -388.268} C_VEL
LIN {X 0,Y 608.43,Z 446.348,A -85,B 0,C 180,E1 -390.547,E2 -390.547} C_VEL
LIN {X 0,Y 608.416,Z 443.119,A -85,B 0,C 180,E1 -392.882,E2 -392.882} C_VEL
LIN {X 0,Y 608.407,Z 440.703,A -85,B 0,C 180,E1 -394.473,E2 -394.473} C_VEL
LIN {X 0,Y 608.482,Z 440.692,A -85,B 0,C 180,E1 -397.16,E2 -397.16} C_VEL
LIN {X 0,Y 608.44,Z 440.699,A -85,B 0,C 180,E1 -399.442,E2 -399.442} C_VEL
LIN {X 0,Y 608.464,Z 440.694,A -85,B 0,C 180,E1 -402.334,E2 -402.334} C_VEL
LIN {X 0,Y 608.459,Z 440.695,A -85,B 0,C 180,E1 -404.796,E2 -404.796} C_VEL
LIN {X 0,Y 608.448,Z 440.697,A -85,B 0,C 180,E1 -407.039,E2 -407.039} C_VEL
LIN {X 0,Y 608.455,Z 440.698,A -85,B 0,C 180,E1 -409.697,E2 -409.697} C_VEL
LIN {X 0,Y 608.467,Z 440.697,A -85,B 0,C 180,E1 -412.253,E2 -412.253} C_VEL
LIN {X 0,Y 608.485,Z 440.853,A -85,B 0,C 180,E1 -414.37,E2 -414.37} C_VEL
LIN {X 0,Y 608.526,Z 448.583,A -85,B 0,C 180,E1 -416.73,E2 -416.73} C_VEL
LIN {X 0,Y 608.538,Z 457.859,A -85,B 0,C 180,E1 -419.459,E2 -419.459} C_VEL
LIN {X 0,Y 608.497,Z 467.127,A -85,B 0,C 180,E1 -422.111,E2 -422.111} C_VEL
LIN {X 0,Y 608.469,Z 476.394,A -85,B 0,C 180,E1 -424.7,E2 -424.7} C_VEL
LIN {X 0,Y 608.48,Z 486.985,A -85,B 0,C 180,E1 -427.595,E2 -427.595} C_VEL
LIN {X 0,Y 608.456,Z 497.577,A -85,B 0,C 180,E1 -430.429,E2 -430.429} C_VEL
LIN {X 0,Y 608.454,Z 508.168,A -85,B 0,C 180,E1 -433.216,E2 -433.216} C_VEL
LIN {X 0,Y 608.461,Z 518.855,A -85,B 0,C 180,E1 -435.987,E2 -435.987} C_VEL
LIN {X 0,Y 608.443,Z 527.53,A -85,B 0,C 180,E1 -438.211,E2 -438.211} C_VEL
LIN {X 0,Y 608.542,Z 542.695,A -85,B 0,C 180,E1 -438.53,E2 -438.53} C_VEL
LIN {X 0,Y 608.526,Z 554.276,A -85,B 0,C 180,E1 -438.894,E2 -438.894} C_VEL
LIN {X 0,Y 608.506,Z 566.92,A -85,B 0,C 180,E1 -439.435,E2 -439.435} C_VEL
LIN {X 0,Y 608.483,Z 577.578,A -85,B 0,C 180,E1 -440.023,E2 -440.023} C_VEL
LIN {X 0,Y 608.483,Z 588.474,A -85,B 0,C 180,E1 -440.778,E2 -440.778} C_VEL
LIN {X 0,Y 608.475,Z 599.111,A -85,B 0,C 180,E1 -441.699,E2 -441.699} C_VEL
LIN {X 0,Y 608.471,Z 606.96,A -85,B 0,C 180,E1 -442.534,E2 -442.534} C_VEL
LIN {X 0,Y 608.461,Z 614.286,A -85,B 0,C 180,E1 -443.484,E2 -443.484} C_VEL
LIN {X 0,Y 608.45,Z 619.866,A -85,B 0,C 180,E1 -444.366,E2 -444.366} C_VEL
LIN {X 0,Y 608.432,Z 624.95,A -85,B 0,C 180,E1 -445.362,E2 -445.362} C_VEL
LIN {X 0,Y 608.449,Z 628.896,A -85,B 0,C 180,E1 -446.358,E2 -446.358} C_VEL
LIN {X 0,Y 608.425,Z 631.809,A -85,B 0,C 180,E1 -447.352,E2 -447.352} C_VEL
LIN {X 0,Y 608.443,Z 633.201,A -85,B 0,C 180,E1 -448.014,E2 -448.014} C_VEL
LIN {X 0,Y 608.438,Z 634.783,A -85,B 0,C 180,E1 -449.338,E2 -449.338} C_VEL
LIN {X 0,Y 608.434,Z 635,A -85,B 0,C 180,E1 -450,E2 -450} C_VEL
LIN {X 0,Y 608.448,Z 634.184,A -85,B 0,C 180,E1 -451.324,E2 -451.324} C_VEL
LIN {X 0,Y 608.443,Z 633.201,A -85,B 0,C 180,E1 -451.986,E2 -451.986} C_VEL
LIN {X 0,Y 608.425,Z 631.809,A -85,B 0,C 180,E1 -452.648,E2 -452.648} C_VEL
LIN {X 0,Y 608.449,Z 628.896,A -85,B 0,C 180,E1 -453.642,E2 -453.642} C_VEL
LIN {X 0,Y 608.432,Z 624.95,A -85,B 0,C 180,E1 -454.638,E2 -454.638} C_VEL
LIN {X 0,Y 608.437,Z 618.876,A -85,B 0,C 180,E1 -455.801,E2 -455.801} C_VEL
LIN {X 0,Y 608.462,Z 612.235,A -85,B 0,C 180,E1 -456.799,E2 -456.799} C_VEL
LIN {X 0,Y 608.455,Z 603.989,A -85,B 0,C 180,E1 -457.8,E2 -457.8} C_VEL
LIN {X 0,Y 608.472,Z 595.536,A -85,B 0,C 180,E1 -458.636,E2 -458.636} C_VEL
LIN {X 0,Y 608.48,Z 585.09,A -85,B 0,C 180,E1 -459.473,E2 -459.473} C_VEL
LIN {X 0,Y 608.494,Z 574.755,A -85,B 0,C 180,E1 -460.145,E2 -460.145} C_VEL
LIN {X 0,Y 608.51,Z 563.265,A -85,B 0,C 180,E1 -460.74,E2 -460.74} C_VEL
LIN {X 0,Y 608.537,Z 550.908,A -85,B 0,C 180,E1 -461.224,E2 -461.224} C_VEL
LIN {X 0,Y 608.543,Z 537.436,A -85,B 0,C 180,E1 -461.597,E2 -461.597} C_VEL
LIN {X 0,Y 608.443,Z 527.53,A -85,B 0,C 180,E1 -461.789,E2 -461.789} C_VEL
LIN {X 0,Y 608.442,Z 517.435,A -85,B 0,C 180,E1 -464.38,E2 -464.38} C_VEL
LIN {X 0,Y 608.447,Z 506.844,A -85,B 0,C 180,E1 -467.13,E2 -467.13} C_VEL
LIN {X 0,Y 608.453,Z 496.253,A -85,B 0,C 180,E1 -469.922,E2 -469.922} C_VEL
LIN {X 0,Y 608.462,Z 485.663,A -85,B 0,C 180,E1 -472.764,E2 -472.764} C_VEL
LIN {X 0,Y 608.469,Z 476.394,A -85,B 0,C 180,E1 -475.3,E2 -475.3} C_VEL
LIN {X 0,Y 608.497,Z 467.127,A -85,B 0,C 180,E1 -477.889,E2 -477.889} C_VEL
LIN {X 0,Y 608.538,Z 457.859,A -85,B 0,C 180,E1 -480.541,E2 -480.541} C_VEL
LIN {X 0,Y 608.522,Z 448.567,A -85,B 0,C 180,E1 -483.271,E2 -483.271} C_VEL
LIN {X 0,Y 608.506,Z 440.958,A -85,B 0,C 180,E1 -485.68,E2 -485.68} C_VEL
LIN {X 0,Y 608.45,Z 440.696,A -85,B 0,C 180,E1 -486.046,E2 -486.046} C_VEL
LIN {X 0,Y 608.472,Z 440.693,A -85,B 0,C 180,E1 -488.588,E2 -488.588} C_VEL
LIN {X 0,Y 608.467,Z 440.697,A -85,B 0,C 180,E1 -491.343,E2 -491.343} C_VEL
LIN {X 0,Y 608.451,Z 440.695,A -85,B 0,C 180,E1 -494.263,E2 -494.263} C_VEL
LIN {X 0,Y 608.458,Z 440.694,A -85,B 0,C 180,E1 -497.04,E2 -497.04} C_VEL
LIN {X 0,Y 608.455,Z 440.696,A -85,B 0,C 180,E1 -499.697,E2 -499.697} C_VEL
LIN {X 0,Y 608.473,Z 440.696,A -85,B 0,C 180,E1 -502.254,E2 -502.254} C_VEL
LIN {X 0,Y 608.412,Z 440.771,A -85,B 0,C 180,E1 -504.72,E2 -504.72} C_VEL
LIN {X 0,Y 608.463,Z 443.953,A -85,B 0,C 180,E1 -507.478,E2 -507.478} C_VEL
LIN {X 0,Y 608.432,Z 447.196,A -85,B 0,C 180,E1 -510.218,E2 -510.218} C_VEL
LIN {X 0,Y 608.427,Z 450.493,A -85,B 0,C 180,E1 -512.803,E2 -512.803} C_VEL
LIN {X 0,Y 608.424,Z 453.921,A -85,B 0,C 180,E1 -515.428,E2 -515.428} C_VEL
LIN {X 0,Y 608.418,Z 457.764,A -85,B 0,C 180,E1 -518.307,E2 -518.307} C_VEL
LIN {X 0,Y 608.434,Z 461.607,A -85,B 0,C 180,E1 -521.13,E2 -521.13} C_VEL
LIN {X 0,Y 608.42,Z 465.451,A -85,B 0,C 180,E1 -523.905,E2 -523.905} C_VEL
LIN {X 0,Y 608.434,Z 469.294,A -85,B 0,C 180,E1 -526.643,E2 -526.643} C_VEL
LIN {X 0,Y 608.429,Z 471.666,A -85,B 0,C 180,E1 -528.317,E2 -528.317} C_VEL
LIN {X 0,Y 608.534,Z 487.515,A -85,B 0,C 180,E1 -528.711,E2 -528.711} C_VEL
LIN {X 0,Y 608.504,Z 500.158,A -85,B 0,C 180,E1 -529.171,E2 -529.171} C_VEL
LIN {X 0,Y 608.48,Z 512.503,A -85,B 0,C 180,E1 -529.771,E2 -529.771} C_VEL
LIN {X 0,Y 608.486,Z 523.306,A -85,B 0,C 180,E1 -530.443,E2 -530.443} C_VEL
LIN {X 0,Y 608.477,Z 533.078,A -85,B 0,C 180,E1 -531.197,E2 -531.197} C_VEL
LIN {X 0,Y 608.46,Z 541.977,A -85,B 0,C 180,E1 -532.033,E2 -532.033} C_VEL
LIN {X 0,Y 608.465,Z 550.664,A -85,B 0,C 180,E1 -533.034,E2 -533.034} C_VEL
LIN {X 0,Y 608.439,Z 557.593,A -85,B 0,C 180,E1 -534.033,E2 -534.033} C_VEL
LIN {X 0,Y 608.436,Z 563.147,A -85,B 0,C 180,E1 -535.03,E2 -535.03} C_VEL
LIN {X 0,Y 608.434,Z 567.509,A -85,B 0,C 180,E1 -536.026,E2 -536.026} C_VEL
LIN {X 0,Y 608.426,Z 569.813,A -85,B 0,C 180,E1 -536.689,E2 -536.689} C_VEL
LIN {X 0,Y 608.425,Z 571.691,A -85,B 0,C 180,E1 -537.352,E2 -537.352} C_VEL
LIN {X 0,Y 608.442,Z 573.127,A -85,B 0,C 180,E1 -538.014,E2 -538.014} C_VEL
LIN {X 0,Y 608.439,Z 574.752,A -85,B 0,C 180,E1 -539.338,E2 -539.338} C_VEL
LIN {X 0,Y 608.434,Z 574.995,A -85,B 0,C 180,E1 -540,E2 -540} C_VEL
LIN {X 0,Y 608.439,Z 574.815,A -85,B 0,C 180,E1 -540.662,E2 -540.662} C_VEL
LIN {X 0,Y 608.441,Z 573.276,A -85,B 0,C 180,E1 -541.986,E2 -541.986} C_VEL
LIN {X 0,Y 608.426,Z 571.918,A -85,B 0,C 180,E1 -542.648,E2 -542.648} C_VEL
LIN {X 0,Y 608.45,Z 569.041,A -85,B 0,C 180,E1 -543.643,E2 -543.643} C_VEL
LIN {X 0,Y 608.433,Z 565.142,A -85,B 0,C 180,E1 -544.638,E2 -544.638} C_VEL
LIN {X 0,Y 608.449,Z 560.111,A -85,B 0,C 180,E1 -545.635,E2 -545.635} C_VEL
LIN {X 0,Y 608.442,Z 553.794,A -85,B 0,C 180,E1 -546.633,E2 -546.633} C_VEL
LIN {X 0,Y 608.475,Z 545.876,A -85,B 0,C 180,E1 -547.633,E2 -547.633} C_VEL
LIN {X 0,Y 608.472,Z 536.034,A -85,B 0,C 180,E1 -548.636,E2 -548.636} C_VEL
LIN {X 0,Y 608.477,Z 533.927,A -85,B 0,C 180,E1 -548.82,E2 -548.82} C_VEL
LIN {X 0,Y 607.803,Z 529.592,A -85,B 0,C 180,E1 -549.19,E2 -549.19} C_VEL
LIN {X 0,Y 604.94,Z 522.346,A -85,B 0,C 180,E1 -549.77,E2 -549.77} C_VEL
LIN {X 0,Y 602.126,Z 514.704,A -85,B 0,C 180,E1 -550.302,E2 -550.302} C_VEL
LIN {X 0,Y 601.531,Z 509.637,A -85,B 0,C 180,E1 -550.595,E2 -550.595} C_VEL
LIN {X 0,Y 601.511,Z 499.137,A -85,B 0,C 180,E1 -551.091,E2 -551.091} C_VEL
LIN {X 0,Y 601.567,Z 486.569,A -85,B 0,C 180,E1 -551.541,E2 -551.541} C_VEL
LIN {X 0,Y 601.491,Z 473.051,A -85,B 0,C 180,E1 -551.868,E2 -551.868} C_VEL
LIN {X 0,Y 601.336,Z 471.643,A -85,B 0,C 180,E1 -551.93,E2 -551.93} C_VEL
LIN {X 0,Y 601.325,Z 468.459,A -85,B 0,C 180,E1 -554.208,E2 -554.208} C_VEL
LIN {X 0,Y 601.338,Z 464.614,A -85,B 0,C 180,E1 -556.989,E2 -556.989} C_VEL
LIN {X 0,Y 601.314,Z 460.768,A -85,B 0,C 180,E1 -559.813,E2 -559.813} C_VEL
LIN {X 0,Y 601.339,Z 457.884,A -85,B 0,C 180,E1 -561.962,E2 -561.962} C_VEL
LIN {X 0,Y 601.343,Z 454.039,A -85,B 0,C 180,E1 -564.882,E2 -564.882} C_VEL
LIN {X 0,Y 601.344,Z 450.858,A -85,B 0,C 180,E1 -567.349,E2 -567.349} C_VEL
LIN {X 0,Y 601.36,Z 447.308,A -85,B 0,C 180,E1 -570.168,E2 -570.168} C_VEL
LIN {X 0,Y 601.361,Z 444.318,A -85,B 0,C 180,E1 -572.706,E2 -572.706} C_VEL
LIN {X 0,Y 601.369,Z 441.58,A -85,B 0,C 180,E1 -575.108,E2 -575.108} C_VEL
LIN {X 0,Y 601.439,Z 441.566,A -85,B 0,C 180,E1 -577.419,E2 -577.419} C_VEL
LIN {X 0,Y 601.404,Z 441.57,A -85,B 0,C 180,E1 -579.996,E2 -579.996} C_VEL
LIN {X 0,Y 601.416,Z 441.568,A -85,B 0,C 180,E1 -582.67,E2 -582.67} C_VEL
LIN {X 0,Y 601.43,Z 441.572,A -85,B 0,C 180,E1 -585.465,E2 -585.465} C_VEL
LIN {X 0,Y 601.426,Z 441.566,A -85,B 0,C 180,E1 -588.407,E2 -588.407} C_VEL
LIN {X 0,Y 601.431,Z 441.57,A -85,B 0,C 180,E1 -590.875,E2 -590.875} C_VEL
LIN {X 0,Y 601.404,Z 441.568,A -85,B 0,C 180,E1 -593.417,E2 -593.417} C_VEL
LIN {X 0,Y 601.438,Z 441.569,A -85,B 0,C 180,E1 -596.064,E2 -596.064} C_VEL
LIN {X 0,Y 601.425,Z 441.566,A -85,B 0,C 180,E1 -598.546,E2 -598.546} C_VEL
LIN {X 0,Y 601.43,Z 441.568,A -85,B 0,C 180,E1 -601.373,E2 -601.373} C_VEL
LIN {X 0,Y 601.404,Z 441.568,A -85,B 0,C 180,E1 -603.636,E2 -603.636} C_VEL
LIN {X 0,Y 601.454,Z 441.566,A -85,B 0,C 180,E1 -605.859,E2 -605.859} C_VEL
LIN {X 0,Y 601.409,Z 441.567,A -85,B 0,C 180,E1 -608.761,E2 -608.761} C_VEL
LIN {X 0,Y 601.429,Z 441.569,A -85,B 0,C 180,E1 -611.608,E2 -611.608} C_VEL
LIN {X 0,Y 601.415,Z 441.57,A -85,B 0,C 180,E1 -614.409,E2 -614.409} C_VEL
LIN {X 0,Y 601.416,Z 441.567,A -85,B 0,C 180,E1 -617.172,E2 -617.172} C_VEL
LIN {X 0,Y 601.436,Z 441.572,A -85,B 0,C 180,E1 -619.905,E2 -619.905} C_VEL
LIN {X 0,Y 601.444,Z 441.564,A -85,B 0,C 180,E1 -622.615,E2 -622.615} C_VEL
LIN {X 0,Y 601.416,Z 441.57,A -85,B 0,C 180,E1 -625.308,E2 -625.308} C_VEL
LIN {X 0,Y 601.437,Z 441.566,A -85,B 0,C 180,E1 -627.991,E2 -627.991} C_VEL
LIN {X 0,Y 601.447,Z 441.564,A -85,B 0,C 180,E1 -630.67,E2 -630.67} C_VEL
LIN {X 0,Y 601.43,Z 441.569,A -85,B 0,C 180,E1 -633.35,E2 -633.35} C_VEL
LIN {X 0,Y 601.416,Z 441.567,A -85,B 0,C 180,E1 -636.037,E2 -636.037} C_VEL
LIN {X 0,Y 601.417,Z 441.574,A -85,B 0,C 180,E1 -638.738,E2 -638.738} C_VEL
LIN {X 0,Y 601.427,Z 441.565,A -85,B 0,C 180,E1 -641.458,E2 -641.458} C_VEL
LIN {X 0,Y 601.426,Z 441.569,A -85,B 0,C 180,E1 -644.205,E2 -644.205} C_VEL
LIN {X 0,Y 601.42,Z 441.569,A -85,B 0,C 180,E1 -646.986,E2 -646.986} C_VEL
LIN {X 0,Y 601.408,Z 441.568,A -85,B 0,C 180,E1 -649.809,E2 -649.809} C_VEL
LIN {X 0,Y 601.418,Z 441.571,A -85,B 0,C 180,E1 -652.683,E2 -652.683} C_VEL
LIN {X 0,Y 601.403,Z 441.569,A -85,B 0,C 180,E1 -654.879,E2 -654.879} C_VEL
LIN {X 0,Y 601.416,Z 441.57,A -85,B 0,C 180,E1 -657.361,E2 -657.361} C_VEL
LIN {X 0,Y 601.433,Z 441.565,A -85,B 0,C 180,E1 -660.164,E2 -660.164} C_VEL
LIN {X 0,Y 601.419,Z 441.573,A -85,B 0,C 180,E1 -662.714,E2 -662.714} C_VEL
LIN {X 0,Y 601.405,Z 441.569,A -85,B 0,C 180,E1 -665.112,E2 -665.112} C_VEL
LIN {X 0,Y 601.437,Z 441.565,A -85,B 0,C 180,E1 -667.419,E2 -667.419} C_VEL
LIN {X 0,Y 601.408,Z 441.571,A -85,B 0,C 180,E1 -669.996,E2 -669.996} C_VEL
LIN {X 0,Y 601.411,Z 441.569,A -85,B 0,C 180,E1 -672.671,E2 -672.671} C_VEL
LIN {X 0,Y 601.432,Z 441.565,A -85,B 0,C 180,E1 -675.482,E2 -675.482} C_VEL
LIN {X 0,Y 601.427,Z 441.571,A -85,B 0,C 180,E1 -678.407,E2 -678.407} C_VEL
LIN {X 0,Y 601.407,Z 441.568,A -85,B 0,C 180,E1 -680.873,E2 -680.873} C_VEL
LIN {X 0,Y 601.405,Z 441.576,A -85,B 0,C 180,E1 -683.417,E2 -683.417} C_VEL
LIN {X 0,Y 601.394,Z 441.577,A -85,B 0,C 180,E1 -685.066,E2 -685.066} C_VEL
LIN {X 0,Y 601.377,Z 442.421,A -85,B 0,C 180,E1 -686.073,E2 -686.073} C_VEL
LIN {X 0,Y 601.372,Z 445.589,A -85,B 0,C 180,E1 -688.553,E2 -688.553} C_VEL
LIN {X 0,Y 601.341,Z 449.118,A -85,B 0,C 180,E1 -691.368,E2 -691.368} C_VEL
LIN {X 0,Y 601.358,Z 452.657,A -85,B 0,C 180,E1 -694.144,E2 -694.144} C_VEL
LIN {X 0,Y 601.333,Z 455.843,A -85,B 0,C 180,E1 -696.586,E2 -696.586} C_VEL
LIN {X 0,Y 601.348,Z 459.686,A -85,B 0,C 180,E1 -699.475,E2 -699.475} C_VEL
LIN {X 0,Y 601.31,Z 463.529,A -85,B 0,C 180,E1 -702.309,E2 -702.309} C_VEL
LIN {X 0,Y 601.317,Z 466.412,A -85,B 0,C 180,E1 -704.406,E2 -704.406} C_VEL
LIN {X 0,Y 601.321,Z 470.255,A -85,B 0,C 180,E1 -707.169,E2 -707.169} C_VEL
LIN {X 0,Y 601.337,Z 471.667,A -85,B 0,C 180,E1 -708.177,E2 -708.177} C_VEL
LIN {X 0,Y 601.599,Z 478.214,A -85,B 0,C 180,E1 -708.331,E2 -708.331} C_VEL
LIN {X 0,Y 601.567,Z 490.85,A -85,B 0,C 180,E1 -708.688,E2 -708.688} C_VEL
LIN {X 0,Y 601.549,Z 503.098,A -85,B 0,C 180,E1 -709.171,E2 -709.171} C_VEL
LIN {X 0,Y 601.474,Z 513.997,A -85,B 0,C 180,E1 -709.735,E2 -709.735} C_VEL
LIN {X 0,Y 601.448,Z 524.459,A -85,B 0,C 180,E1 -710.415,E2 -710.415} C_VEL
LIN {X 0,Y 601.436,Z 535.009,A -85,B 0,C 180,E1 -711.262,E2 -711.262} C_VEL
LIN {X 0,Y 601.4,Z 543.588,A -85,B 0,C 180,E1 -712.108,E2 -712.108} C_VEL
LIN {X 0,Y 601.388,Z 551.905,A -85,B 0,C 180,E1 -713.12,E2 -713.12} C_VEL
LIN {X 0,Y 601.373,Z 558.605,A -85,B 0,C 180,E1 -714.131,E2 -714.131} C_VEL
LIN {X 0,Y 601.335,Z 564.747,A -85,B 0,C 180,E1 -715.307,E2 -715.307} C_VEL
LIN {X 0,Y 601.368,Z 568.737,A -85,B 0,C 180,E1 -716.314,E2 -716.314} C_VEL
LIN {X 0,Y 601.325,Z 571.688,A -85,B 0,C 180,E1 -717.32,E2 -717.32} C_VEL
LIN {X 0,Y 601.341,Z 573.123,A -85,B 0,C 180,E1 -717.991,E2 -717.991} C_VEL
LIN {X 0,Y 601.34,Z 574.752,A -85,B 0,C 180,E1 -719.33,E2 -719.33} C_VEL
LIN {X 0,Y 601.335,Z 574.99,A -85,B 0,C 180,E1 -720,E2 -720} C_VEL
LIN {X 0,Y 601.339,Z 574.814,A -85,B 0,C 180,E1 -720.669,E2 -720.669} C_VEL
LIN {X 0,Y 601.349,Z 574.238,A -85,B 0,C 180,E1 -721.339,E2 -721.339} C_VEL
LIN {X 0,Y 601.326,Z 571.917,A -85,B 0,C 180,E1 -722.679,E2 -722.679} C_VEL
LIN {X 0,Y 601.369,Z 569.043,A -85,B 0,C 180,E1 -723.685,E2 -723.685} C_VEL
LIN {X 0,Y 601.337,Z 565.143,A -85,B 0,C 180,E1 -724.693,E2 -724.693} C_VEL
LIN {X 0,Y 601.373,Z 560.11,A -85,B 0,C 180,E1 -725.701,E2 -725.701} C_VEL
LIN {X 0,Y 601.382,Z 553.781,A -85,B 0,C 180,E1 -726.711,E2 -726.711} C_VEL
LIN {X 0,Y 601.396,Z 545.879,A -85,B 0,C 180,E1 -727.723,E2 -727.723} C_VEL
LIN {X 0,Y 601.436,Z 536.03,A -85,B 0,C 180,E1 -728.738,E2 -728.738} C_VEL
LIN {X 0,Y 601.446,Z 525.7,A -85,B 0,C 180,E1 -729.585,E2 -729.585} C_VEL
LIN {X 0,Y 601.471,Z 515.501,A -85,B 0,C 180,E1 -730.264,E2 -730.264} C_VEL
LIN {X 0,Y 601.515,Z 503.839,A -85,B 0,C 180,E1 -730.884,E2 -730.884} C_VEL
LIN {X 0,Y 601.56,Z 491.617,A -85,B 0,C 180,E1 -731.377,E2 -731.377} C_VEL
LIN {X 0,Y 601.606,Z 479.334,A -85,B 0,C 180,E1 -731.732,E2 -731.732} C_VEL
LIN {X 0,Y 601.358,Z 472.233,A -85,B 0,C 180,E1 -731.887,E2 -731.887} C_VEL
LIN {X 0,Y 601.34,Z 471.643,A -85,B 0,C 180,E1 -731.93,E2 -731.93} C_VEL
LIN {X 0,Y 601.319,Z 468.459,A -85,B 0,C 180,E1 -734.208,E2 -734.208} C_VEL
LIN {X 0,Y 601.338,Z 464.614,A -85,B 0,C 180,E1 -736.989,E2 -736.989} C_VEL
LIN {X 0,Y 601.315,Z 460.769,A -85,B 0,C 180,E1 -739.812,E2 -739.812} C_VEL
LIN {X 0,Y 601.338,Z 457.885,A -85,B 0,C 180,E1 -741.962,E2 -741.962} C_VEL
LIN {X 0,Y 601.345,Z 454.039,A -85,B 0,C 180,E1 -744.881,E2 -744.881} C_VEL
LIN {X 0,Y 601.344,Z 450.858,A -85,B 0,C 180,E1 -747.349,E2 -747.349} C_VEL
LIN {X 0,Y 601.359,Z 447.309,A -85,B 0,C 180,E1 -750.168,E2 -750.168} C_VEL
LIN {X 0,Y 601.345,Z 443.952,A -85,B 0,C 180,E1 -752.521,E2 -752.521} C_VEL
LIN {X 0,Y 601.324,Z 441.585,A -85,B 0,C 180,E1 -754.125,E2 -754.125} C_VEL
LIN {X 0,Y 601.407,Z 441.572,A -85,B 0,C 180,E1 -756.583,E2 -756.583} C_VEL
LIN {X 0,Y 601.405,Z 441.572,A -85,B 0,C 180,E1 -759.127,E2 -759.127} C_VEL
LIN {X 0,Y 601.43,Z 441.57,A -85,B 0,C 180,E1 -761.765,E2 -761.765} C_VEL
LIN {X 0,Y 601.428,Z 441.572,A -85,B 0,C 180,E1 -764.535,E2 -764.535} C_VEL
LIN {X 0,Y 601.409,Z 441.573,A -85,B 0,C 180,E1 -767.41,E2 -767.41} C_VEL
LIN {X 0,Y 601.445,Z 441.567,A -85,B 0,C 180,E1 -770.464,E2 -770.464} C_VEL
LIN {X 0,Y 601.403,Z 441.576,A -85,B 0,C 180,E1 -773.417,E2 -773.417} C_VEL
LIN {X 0,Y 601.457,Z 441.73,A -85,B 0,C 180,E1 -774.16,E2 -774.16} C_VEL
LIN {X 0,Y 601.586,Z 447.751,A -85,B 0,C 180,E1 -776.043,E2 -776.043} C_VEL
LIN {X 0,Y 601.548,Z 456.015,A -85,B 0,C 180,E1 -778.526,E2 -778.526} C_VEL
LIN {X 0,Y 601.504,Z 465.19,A -85,B 0,C 180,E1 -781.2,E2 -781.2} C_VEL
LIN {X 0,Y 601.475,Z 473.746,A -85,B 0,C 180,E1 -783.64,E2 -783.64} C_VEL
LIN {X 0,Y 601.46,Z 483.014,A -85,B 0,C 180,E1 -786.226,E2 -786.226} C_VEL
LIN {X 0,Y 601.442,Z 492.281,A -85,B 0,C 180,E1 -788.762,E2 -788.762} C_VEL
LIN {X 0,Y 601.401,Z 502.872,A -85,B 0,C 180,E1 -791.608,E2 -791.608} C_VEL
LIN {X 0,Y 601.385,Z 513.464,A -85,B 0,C 180,E1 -794.408,E2 -794.408} C_VEL
LIN {X 0,Y 601.362,Z 524.055,A -85,B 0,C 180,E1 -797.171,E2 -797.171} C_VEL
LIN {X 0,Y 601.387,Z 527.53,A -85,B 0,C 180,E1 -798.071,E2 -798.071} C_VEL
LIN {X 0,Y 601.601,Z 540.179,A -85,B 0,C 180,E1 -798.332,E2 -798.332} C_VEL
LIN {X 0,Y 601.568,Z 552.204,A -85,B 0,C 180,E1 -798.687,E2 -798.687} C_VEL
LIN {X 0,Y 601.511,Z 564.017,A -85,B 0,C 180,E1 -799.169,E2 -799.169} C_VEL
LIN {X 0,Y 601.494,Z 576.167,A -85,B 0,C 180,E1 -799.821,E2 -799.821} C_VEL
LIN {X 0,Y 601.455,Z 587.402,A -85,B 0,C 180,E1 -800.585,E2 -800.585} C_VEL
LIN {X 0,Y 601.423,Z 597.336,A -85,B 0,C 180,E1 -801.431,E2 -801.431} C_VEL
LIN {X 0,Y 601.418,Z 606.96,A -85,B 0,C 180,E1 -802.446,E2 -802.446} C_VEL
LIN {X 0,Y 601.37,Z 614.224,A -85,B 0,C 180,E1 -803.398,E2 -803.398} C_VEL
LIN {X 0,Y 601.372,Z 619.866,A -85,B 0,C 180,E1 -804.299,E2 -804.299} C_VEL
LIN {X 0,Y 601.337,Z 624.95,A -85,B 0,C 180,E1 -805.307,E2 -805.307} C_VEL
LIN {X 0,Y 601.367,Z 628.896,A -85,B 0,C 180,E1 -806.315,E2 -806.315} C_VEL
LIN {X 0,Y 601.325,Z 631.809,A -85,B 0,C 180,E1 -807.32,E2 -807.32} C_VEL
LIN {X 0,Y 601.341,Z 633.202,A -85,B 0,C 180,E1 -807.991,E2 -807.991} C_VEL
LIN {X 0,Y 601.339,Z 634.784,A -85,B 0,C 180,E1 -809.33,E2 -809.33} C_VEL
LIN {X 0,Y 601.335,Z 635,A -85,B 0,C 180,E1 -810,E2 -810} C_VEL
LIN {X 0,Y 601.348,Z 634.184,A -85,B 0,C 180,E1 -811.339,E2 -811.339} C_VEL
LIN {X 0,Y 601.341,Z 633.202,A -85,B 0,C 180,E1 -812.009,E2 -812.009} C_VEL
LIN {X 0,Y 601.325,Z 631.809,A -85,B 0,C 180,E1 -812.68,E2 -812.68} C_VEL
LIN {X 0,Y 601.367,Z 628.896,A -85,B 0,C 180,E1 -813.685,E2 -813.685} C_VEL
LIN {X 0,Y 601.337,Z 624.95,A -85,B 0,C 180,E1 -814.693,E2 -814.693} C_VEL
LIN {X 0,Y 601.372,Z 618.877,A -85,B 0,C 180,E1 -815.869,E2 -815.869} C_VEL
LIN {X 0,Y 601.382,Z 612.235,A -85,B 0,C 180,E1 -816.88,E2 -816.88} C_VEL
LIN {X 0,Y 601.4,Z 603.989,A -85,B 0,C 180,E1 -817.892,E2 -817.892} C_VEL
LIN {X 0,Y 601.436,Z 595.536,A -85,B 0,C 180,E1 -818.738,E2 -818.738} C_VEL
LIN {X 0,Y 601.449,Z 585.091,A -85,B 0,C 180,E1 -819.585,E2 -819.585} C_VEL
LIN {X 0,Y 601.472,Z 574.756,A -85,B 0,C 180,E1 -820.264,E2 -820.264} C_VEL
LIN {X 0,Y 601.534,Z 562.636,A -85,B 0,C 180,E1 -820.894,E2 -820.894} C_VEL
LIN {X 0,Y 601.569,Z 550.223,A -85,B 0,C 180,E1 -821.378,E2 -821.378} C_VEL
LIN {X 0,Y 601.599,Z 537.435,A -85,B 0,C 180,E1 -821.733,E2 -821.733} C_VEL
LIN {X 0,Y 601.387,Z 527.53,A -85,B 0,C 180,E1 -821.929,E2 -821.929} C_VEL
LIN {X 0,Y 601.39,Z 517.435,A -85,B 0,C 180,E1 -824.552,E2 -824.552} C_VEL
LIN {X 0,Y 601.389,Z 506.844,A -85,B 0,C 180,E1 -827.338,E2 -827.338} C_VEL
LIN {X 0,Y 601.424,Z 496.253,A -85,B 0,C 180,E1 -830.165,E2 -830.165} C_VEL
LIN {X 0,Y 601.431,Z 485.661,A -85,B 0,C 180,E1 -833.046,E2 -833.046} C_VEL
LIN {X 0,Y 601.471,Z 476.394,A -85,B 0,C 180,E1 -835.616,E2 -835.616} C_VEL
LIN {X 0,Y 601.495,Z 467.127,A -85,B 0,C 180,E1 -838.243,E2 -838.243} C_VEL
LIN {X 0,Y 601.544,Z 457.859,A -85,B 0,C 180,E1 -840.935,E2 -840.935} C_VEL
LIN {X 0,Y 601.561,Z 449.839,A -85,B 0,C 180,E1 -843.305,E2 -843.305} C_VEL
LIN {X 0,Y 601.598,Z 444.091,A -85,B 0,C 180,E1 -845.139,E2 -845.139} C_VEL
LIN {X 0,Y 601.423,Z 441.573,A -85,B 0,C 180,E1 -846.023,E2 -846.023} C_VEL
LIN {X 0,Y 601.435,Z 441.569,A -85,B 0,C 180,E1 -848.471,E2 -848.471} C_VEL
LIN {X 0,Y 601.422,Z 441.571,A -85,B 0,C 180,E1 -850.874,E2 -850.874} C_VEL
LIN {X 0,Y 601.431,Z 441.571,A -85,B 0,C 180,E1 -853.586,E2 -853.586} C_VEL
LIN {X 0,Y 601.454,Z 441.568,A -85,B 0,C 180,E1 -856.425,E2 -856.425} C_VEL
LIN {X 0,Y 601.417,Z 441.571,A -85,B 0,C 180,E1 -859.427,E2 -859.427} C_VEL
LIN {X 0,Y 601.426,Z 441.57,A -85,B 0,C 180,E1 -861.732,E2 -861.732} C_VEL
LIN {X 0,Y 601.379,Z 441.576,A -85,B 0,C 180,E1 -864.245,E2 -864.245} C_VEL
LIN {X 0,Y 601.393,Z 441.893,A -85,B 0,C 180,E1 -865.067,E2 -865.067} C_VEL
LIN {X 0,Y 601.398,Z 444.658,A -85,B 0,C 180,E1 -867.482,E2 -867.482} C_VEL
LIN {X 0,Y 601.355,Z 447.255,A -85,B 0,C 180,E1 -869.864,E2 -869.864} C_VEL
LIN {X 0,Y 601.346,Z 450.743,A -85,B 0,C 180,E1 -872.651,E2 -872.651} C_VEL
LIN {X 0,Y 601.346,Z 453.922,A -85,B 0,C 180,E1 -875.119,E2 -875.119} C_VEL
LIN {X 0,Y 601.339,Z 457.765,A -85,B 0,C 180,E1 -878.038,E2 -878.038} C_VEL
LIN {X 0,Y 601.315,Z 460.647,A -85,B 0,C 180,E1 -880.188,E2 -880.188} C_VEL
LIN {X 0,Y 601.337,Z 464.491,A -85,B 0,C 180,E1 -883.011,E2 -883.011} C_VEL
LIN {X 0,Y 601.338,Z 468.541,A -85,B 0,C 180,E1 -885.941,E2 -885.941} C_VEL
LIN {X 0,Y 601.336,Z 471.667,A -85,B 0,C 180,E1 -888.177,E2 -888.177} C_VEL
LIN {X 0,Y 601.584,Z 477.344,A -85,B 0,C 180,E1 -888.31,E2 -888.31} C_VEL
LIN {X 0,Y 601.558,Z 490.059,A -85,B 0,C 180,E1 -888.661,E2 -888.661} C_VEL
LIN {X 0,Y 601.527,Z 501.687,A -85,B 0,C 180,E1 -889.109,E2 -889.109} C_VEL
LIN {X 0,Y 601.493,Z 512.514,A -85,B 0,C 180,E1 -889.651,E2 -889.651} C_VEL
LIN {X 0,Y 601.46,Z 523.312,A -85,B 0,C 180,E1 -890.33,E2 -890.33} C_VEL
LIN {X 0,Y 601.435,Z 533.085,A -85,B 0,C 180,E1 -891.093,E2 -891.093} C_VEL
LIN {X 0,Y 601.407,Z 541.982,A -85,B 0,C 180,E1 -891.939,E2 -891.939} C_VEL
LIN {X 0,Y 601.407,Z 550.668,A -85,B 0,C 180,E1 -892.952,E2 -892.952} C_VEL
LIN {X 0,Y 601.361,Z 557.597,A -85,B 0,C 180,E1 -893.963,E2 -893.963} C_VEL
LIN {X 0,Y 601.345,Z 563.15,A -85,B 0,C 180,E1 -894.971,E2 -894.971} C_VEL
LIN {X 0,Y 601.346,Z 567.511,A -85,B 0,C 180,E1 -895.979,E2 -895.979} C_VEL
LIN {X 0,Y 601.345,Z 569.815,A -85,B 0,C 180,E1 -896.65,E2 -896.65} C_VEL
LIN {X 0,Y 601.324,Z 571.693,A -85,B 0,C 180,E1 -897.321,E2 -897.321} C_VEL
LIN {X 0,Y 601.341,Z 573.127,A -85,B 0,C 180,E1 -897.991,E2 -897.991} C_VEL
LIN {X 0,Y 601.339,Z 574.753,A -85,B 0,C 180,E1 -899.331,E2 -899.331} C_VEL
LIN {X 0,Y 601.335,Z 574.996,A -85,B 0,C 180,E1 -900,E2 -900} C_VEL
LIN {X 0,Y 601.339,Z 574.815,A -85,B 0,C 180,E1 -900.67,E2 -900.67} C_VEL
LIN {X 0,Y 601.34,Z 573.275,A -85,B 0,C 180,E1 -902.009,E2 -902.009} C_VEL
LIN {X 0,Y 601.326,Z 571.916,A -85,B 0,C 180,E1 -902.68,E2 -902.68} C_VEL
LIN {X 0,Y 601.368,Z 569.039,A -85,B 0,C 180,E1 -903.686,E2 -903.686} C_VEL
LIN {X 0,Y 601.337,Z 565.14,A -85,B 0,C 180,E1 -904.693,E2 -904.693} C_VEL
LIN {X 0,Y 601.373,Z 560.108,A -85,B 0,C 180,E1 -905.701,E2 -905.701} C_VEL
LIN {X 0,Y 601.383,Z 553.79,A -85,B 0,C 180,E1 -906.711,E2 -906.711} C_VEL
LIN {X 0,Y 601.396,Z 545.872,A -85,B 0,C 180,E1 -907.724,E2 -907.724} C_VEL
LIN {X 0,Y 601.437,Z 536.028,A -85,B 0,C 180,E1 -908.738,E2 -908.738} C_VEL
LIN {X 0,Y 601.449,Z 525.705,A -85,B 0,C 180,E1 -909.585,E2 -909.585} C_VEL
LIN {X 0,Y 601.493,Z 514.086,A -85,B 0,C 180,E1 -910.349,E2 -910.349} C_VEL
LIN {X 0,Y 601.531,Z 509.637,A -85,B 0,C 180,E1 -910.595,E2 -910.595} C_VEL
LIN {X 0,Y 600.912,Z 504.501,A -85,B 0,C 180,E1 -910.869,E2 -910.869} C_VEL
LIN {X 0,Y 598.031,Z 496.061,A -85,B 0,C 180,E1 -911.29,E2 -911.29} C_VEL
LIN {X 0,Y 595.196,Z 487.321,A -85,B 0,C 180,E1 -911.645,E2 -911.645} C_VEL
LIN {X 0,Y 594.64,Z 481.725,A -85,B 0,C 180,E1 -911.814,E2 -911.814} C_VEL
LIN {X 0,Y 594.529,Z 473.735,A -85,B 0,C 180,E1 -911.996,E2 -911.996} C_VEL
LIN {X 0,Y 594.24,Z 471.672,A -85,B 0,C 180,E1 -912.053,E2 -912.053} C_VEL
LIN {X 0,Y 594.242,Z 468.458,A -85,B 0,C 180,E1 -914.381,E2 -914.381} C_VEL
LIN {X 0,Y 594.238,Z 464.613,A -85,B 0,C 180,E1 -917.198,E2 -917.198} C_VEL
LIN {X 0,Y 594.246,Z 461.729,A -85,B 0,C 180,E1 -919.339,E2 -919.339} C_VEL
LIN {X 0,Y 594.224,Z 458.845,A -85,B 0,C 180,E1 -921.509,E2 -921.509} C_VEL
LIN {X 0,Y 594.278,Z 454.999,A -85,B 0,C 180,E1 -924.451,E2 -924.451} C_VEL
LIN {X 0,Y 594.258,Z 452.115,A -85,B 0,C 180,E1 -926.706,E2 -926.706} C_VEL
LIN {X 0,Y 594.258,Z 449.232,A -85,B 0,C 180,E1 -929.005,E2 -929.005} C_VEL
LIN {X 0,Y 594.307,Z 446.173,A -85,B 0,C 180,E1 -931.631,E2 -931.631} C_VEL
LIN {X 0,Y 594.294,Z 442.658,A -85,B 0,C 180,E1 -934.586,E2 -934.586} C_VEL
LIN {X 0,Y 594.387,Z 442.448,A -85,B 0,C 180,E1 -937.087,E2 -937.087} C_VEL
LIN {X 0,Y 594.359,Z 442.446,A -85,B 0,C 180,E1 -939.772,E2 -939.772} C_VEL
LIN {X 0,Y 594.374,Z 442.448,A -85,B 0,C 180,E1 -942.375,E2 -942.375} C_VEL
LIN {X 0,Y 594.369,Z 442.447,A -85,B 0,C 180,E1 -945.191,E2 -945.191} C_VEL
LIN {X 0,Y 594.384,Z 442.443,A -85,B 0,C 180,E1 -948.152,E2 -948.152} C_VEL
LIN {X 0,Y 594.384,Z 442.444,A -85,B 0,C 180,E1 -951.195,E2 -951.195} C_VEL
LIN {X 0,Y 594.356,Z 442.449,A -85,B 0,C 180,E1 -953.756,E2 -953.756} C_VEL
LIN {X 0,Y 594.382,Z 442.445,A -85,B 0,C 180,E1 -956.239,E2 -956.239} C_VEL
LIN {X 0,Y 594.375,Z 442.444,A -85,B 0,C 180,E1 -958.65,E2 -958.65} C_VEL
LIN {X 0,Y 594.388,Z 442.45,A -85,B 0,C 180,E1 -961.042,E2 -961.042} C_VEL
LIN {X 0,Y 594.393,Z 442.443,A -85,B 0,C 180,E1 -963.977,E2 -963.977} C_VEL
LIN {X 0,Y 594.378,Z 442.449,A -85,B 0,C 180,E1 -966.295,E2 -966.295} C_VEL
LIN {X 0,Y 594.41,Z 442.442,A -85,B 0,C 180,E1 -969.225,E2 -969.225} C_VEL
LIN {X 0,Y 594.359,Z 442.446,A -85,B 0,C 180,E1 -972.095,E2 -972.095} C_VEL
LIN {X 0,Y 594.368,Z 442.446,A -85,B 0,C 180,E1 -974.219,E2 -974.219} C_VEL
LIN {X 0,Y 594.386,Z 442.448,A -85,B 0,C 180,E1 -976.321,E2 -976.321} C_VEL
LIN {X 0,Y 594.377,Z 442.443,A -85,B 0,C 180,E1 -979.095,E2 -979.095} C_VEL
LIN {X 0,Y 594.417,Z 442.443,A -85,B 0,C 180,E1 -981.843,E2 -981.843} C_VEL
LIN {X 0,Y 594.393,Z 442.444,A -85,B 0,C 180,E1 -984.572,E2 -984.572} C_VEL
LIN {X 0,Y 594.405,Z 442.441,A -85,B 0,C 180,E1 -987.289,E2 -987.289} C_VEL
LIN {X 0,Y 594.42,Z 442.443,A -85,B 0,C 180,E1 -990,E2 -990} C_VEL
LIN {X 0,Y 594.404,Z 442.44,A -85,B 0,C 180,E1 -992.711,E2 -992.711} C_VEL
LIN {X 0,Y 594.401,Z 442.447,A -85,B 0,C 180,E1 -995.428,E2 -995.428} C_VEL
LIN {X 0,Y 594.389,Z 442.443,A -85,B 0,C 180,E1 -998.157,E2 -998.157} C_VEL
LIN {X 0,Y 594.396,Z 442.442,A -85,B 0,C 180,E1 -1001.074,E2 -1001.074} C_VEL
LIN {X 0,Y 594.386,Z 442.447,A -85,B 0,C 180,E1 -1003.679,E2 -1003.679} C_VEL
LIN {X 0,Y 594.376,Z 442.444,A -85,B 0,C 180,E1 -1006.711,E2 -1006.711} C_VEL
LIN {X 0,Y 594.372,Z 442.448,A -85,B 0,C 180,E1 -1009.334,E2 -1009.334} C_VEL
LIN {X 0,Y 594.37,Z 442.445,A -85,B 0,C 180,E1 -1011.503,E2 -1011.503} C_VEL
LIN {X 0,Y 594.395,Z 442.445,A -85,B 0,C 180,E1 -1014.446,E2 -1014.446} C_VEL
LIN {X 0,Y 594.384,Z 442.442,A -85,B 0,C 180,E1 -1016.7,E2 -1016.7} C_VEL
LIN {X 0,Y 594.387,Z 442.445,A -85,B 0,C 180,E1 -1018.998,E2 -1018.998} C_VEL
LIN {X 0,Y 594.389,Z 442.443,A -85,B 0,C 180,E1 -1021.643,E2 -1021.643} C_VEL
LIN {X 0,Y 594.39,Z 442.449,A -85,B 0,C 180,E1 -1024.579,E2 -1024.579} C_VEL
LIN {X 0,Y 594.392,Z 442.445,A -85,B 0,C 180,E1 -1027.608,E2 -1027.608} C_VEL
LIN {X 0,Y 594.368,Z 442.445,A -85,B 0,C 180,E1 -1030.567,E2 -1030.567} C_VEL
LIN {X 0,Y 594.371,Z 442.449,A -85,B 0,C 180,E1 -1033.299,E2 -1033.299} C_VEL
LIN {X 0,Y 594.388,Z 442.445,A -85,B 0,C 180,E1 -1036.159,E2 -1036.159} C_VEL
LIN {X 0,Y 594.379,Z 442.443,A -85,B 0,C 180,E1 -1039.178,E2 -1039.178} C_VEL
LIN {X 0,Y 594.387,Z 442.445,A -85,B 0,C 180,E1 -1042.059,E2 -1042.059} C_VEL
LIN {X 0,Y 594.352,Z 442.449,A -85,B 0,C 180,E1 -1044.677,E2 -1044.677} C_VEL
LIN {X 0,Y 594.288,Z 442.669,A -85,B 0,C 180,E1 -1045.875,E2 -1045.875} C_VEL
LIN {X 0,Y 594.288,Z 446.179,A -85,B 0,C 180,E1 -1048.645,E2 -1048.645} C_VEL
LIN {X 0,Y 594.259,Z 449.205,A -85,B 0,C 180,E1 -1051.064,E2 -1051.064} C_VEL
LIN {X 0,Y 594.259,Z 452.001,A -85,B 0,C 180,E1 -1053.294,E2 -1053.294} C_VEL
LIN {X 0,Y 594.281,Z 454.936,A -85,B 0,C 180,E1 -1055.59,E2 -1055.59} C_VEL
LIN {X 0,Y 594.225,Z 458.726,A -85,B 0,C 180,E1 -1058.491,E2 -1058.491} C_VEL
LIN {X 0,Y 594.243,Z 462.212,A -85,B 0,C 180,E1 -1061.111,E2 -1061.111} C_VEL
LIN {X 0,Y 594.249,Z 465.452,A -85,B 0,C 180,E1 -1063.51,E2 -1063.51} C_VEL
LIN {X 0,Y 594.247,Z 469.295,A -85,B 0,C 180,E1 -1066.318,E2 -1066.318} C_VEL
LIN {X 0,Y 594.263,Z 471.668,A -85,B 0,C 180,E1 -1068.034,E2 -1068.034} C_VEL
LIN {X 0,Y 594.638,Z 477.296,A -85,B 0,C 180,E1 -1068.171,E2 -1068.171} C_VEL
LIN {X 0,Y 594.621,Z 489.088,A -85,B 0,C 180,E1 -1068.495,E2 -1068.495} C_VEL
LIN {X 0,Y 594.535,Z 501.541,A -85,B 0,C 180,E1 -1068.973,E2 -1068.973} C_VEL
LIN {X 0,Y 594.487,Z 514.002,A -85,B 0,C 180,E1 -1069.613,E2 -1069.613} C_VEL
LIN {X 0,Y 594.434,Z 524.459,A -85,B 0,C 180,E1 -1070.3,E2 -1070.3} C_VEL
LIN {X 0,Y 594.382,Z 535.009,A -85,B 0,C 180,E1 -1071.158,E2 -1071.158} C_VEL
LIN {X 0,Y 594.359,Z 543.593,A -85,B 0,C 180,E1 -1072.013,E2 -1072.013} C_VEL
LIN {X 0,Y 594.32,Z 551.91,A -85,B 0,C 180,E1 -1073.038,E2 -1073.038} C_VEL
LIN {X 0,Y 594.305,Z 558.608,A -85,B 0,C 180,E1 -1074.061,E2 -1074.061} C_VEL
LIN {X 0,Y 594.24,Z 564.742,A -85,B 0,C 180,E1 -1075.251,E2 -1075.251} C_VEL
LIN {X 0,Y 594.289,Z 568.734,A -85,B 0,C 180,E1 -1076.271,E2 -1076.271} C_VEL
LIN {X 0,Y 594.225,Z 571.687,A -85,B 0,C 180,E1 -1077.288,E2 -1077.288} C_VEL
LIN {X 0,Y 594.24,Z 573.117,A -85,B 0,C 180,E1 -1077.967,E2 -1077.967} C_VEL
LIN {X 0,Y 594.247,Z 574.134,A -85,B 0,C 180,E1 -1078.644,E2 -1078.644} C_VEL
LIN {X 0,Y 594.236,Z 574.984,A -85,B 0,C 180,E1 -1080,E2 -1080} C_VEL
LIN {X 0,Y 594.239,Z 574.812,A -85,B 0,C 180,E1 -1080.677,E2 -1080.677} C_VEL
LIN {X 0,Y 594.249,Z 574.239,A -85,B 0,C 180,E1 -1081.355,E2 -1081.355} C_VEL
LIN {X 0,Y 594.226,Z 571.914,A -85,B 0,C 180,E1 -1082.711,E2 -1082.711} C_VEL
LIN {X 0,Y 594.29,Z 569.042,A -85,B 0,C 180,E1 -1083.729,E2 -1083.729} C_VEL
LIN {X 0,Y 594.242,Z 565.142,A -85,B 0,C 180,E1 -1084.749,E2 -1084.749} C_VEL
LIN {X 0,Y 594.299,Z 560.103,A -85,B 0,C 180,E1 -1085.769,E2 -1085.769} C_VEL
LIN {X 0,Y 594.316,Z 553.769,A -85,B 0,C 180,E1 -1086.791,E2 -1086.791} C_VEL
LIN {X 0,Y 594.346,Z 545.877,A -85,B 0,C 180,E1 -1087.815,E2 -1087.815} C_VEL
LIN {X 0,Y 594.381,Z 536.02,A -85,B 0,C 180,E1 -1088.842,E2 -1088.842} C_VEL
LIN {X 0,Y 594.425,Z 525.688,A -85,B 0,C 180,E1 -1089.699,E2 -1089.699} C_VEL
LIN {X 0,Y 594.486,Z 515.491,A -85,B 0,C 180,E1 -1090.386,E2 -1090.386} C_VEL
LIN {X 0,Y 594.532,Z 503.404,A -85,B 0,C 180,E1 -1091.034,E2 -1091.034} C_VEL
LIN {X 0,Y 594.589,Z 490.477,A -85,B 0,C 180,E1 -1091.549,E2 -1091.549} C_VEL
LIN {X 0,Y 594.636,Z 477.463,A -85,B 0,C 180,E1 -1091.915,E2 -1091.915} C_VEL
LIN {X 0,Y 594.313,Z 472.215,A -85,B 0,C 180,E1 -1092.03,E2 -1092.03} C_VEL
LIN {X 0,Y 594.253,Z 471.643,A -85,B 0,C 180,E1 -1092.074,E2 -1092.074} C_VEL
LIN {X 0,Y 594.238,Z 468.459,A -85,B 0,C 180,E1 -1094.381,E2 -1094.381} C_VEL
LIN {X 0,Y 594.239,Z 464.613,A -85,B 0,C 180,E1 -1097.198,E2 -1097.198} C_VEL
LIN {X 0,Y 594.241,Z 461.729,A -85,B 0,C 180,E1 -1099.339,E2 -1099.339} C_VEL
LIN {X 0,Y 594.226,Z 458.845,A -85,B 0,C 180,E1 -1101.509,E2 -1101.509} C_VEL
LIN {X 0,Y 594.278,Z 455,A -85,B 0,C 180,E1 -1104.451,E2 -1104.451} C_VEL
LIN {X 0,Y 594.264,Z 452.115,A -85,B 0,C 180,E1 -1106.705,E2 -1106.705} C_VEL
LIN {X 0,Y 594.257,Z 449.231,A -85,B 0,C 180,E1 -1109.005,E2 -1109.005} C_VEL
LIN {X 0,Y 594.257,Z 445.664,A -85,B 0,C 180,E1 -1111.623,E2 -1111.623} C_VEL
LIN {X 0,Y 594.244,Z 442.468,A -85,B 0,C 180,E1 -1113.77,E2 -1113.77} C_VEL
LIN {X 0,Y 594.356,Z 442.45,A -85,B 0,C 180,E1 -1116.244,E2 -1116.244} C_VEL
LIN {X 0,Y 594.373,Z 442.448,A -85,B 0,C 180,E1 -1118.806,E2 -1118.806} C_VEL
LIN {X 0,Y 594.388,Z 442.448,A -85,B 0,C 180,E1 -1121.849,E2 -1121.849} C_VEL
LIN {X 0,Y 594.385,Z 442.447,A -85,B 0,C 180,E1 -1124.236,E2 -1124.236} C_VEL
LIN {X 0,Y 594.361,Z 442.453,A -85,B 0,C 180,E1 -1127.148,E2 -1127.148} C_VEL
LIN {X 0,Y 594.372,Z 442.449,A -85,B 0,C 180,E1 -1129.433,E2 -1129.433} C_VEL
LIN {X 0,Y 594.391,Z 442.449,A -85,B 0,C 180,E1 -1132.392,E2 -1132.392} C_VEL
LIN {X 0,Y 594.391,Z 442.525,A -85,B 0,C 180,E1 -1133.915,E2 -1133.915} C_VEL
LIN {X 0,Y 594.64,Z 447.249,A -85,B 0,C 180,E1 -1135.437,E2 -1135.437} C_VEL
LIN {X 0,Y 594.599,Z 455.106,A -85,B 0,C 180,E1 -1137.867,E2 -1137.867} C_VEL
LIN {X 0,Y 594.556,Z 464.479,A -85,B 0,C 180,E1 -1140.623,E2 -1140.623} C_VEL
LIN {X 0,Y 594.509,Z 473.746,A -85,B 0,C 180,E1 -1143.306,E2 -1143.306} C_VEL
LIN {X 0,Y 594.447,Z 484.338,A -85,B 0,C 180,E1 -1146.298,E2 -1146.298} C_VEL
LIN {X 0,Y 594.405,Z 494.929,A -85,B 0,C 180,E1 -1149.224,E2 -1149.224} C_VEL
LIN {X 0,Y 594.36,Z 505.52,A -85,B 0,C 180,E1 -1152.095,E2 -1152.095} C_VEL
LIN {X 0,Y 594.324,Z 516.111,A -85,B 0,C 180,E1 -1154.921,E2 -1154.921} C_VEL
LIN {X 0,Y 594.295,Z 526.703,A -85,B 0,C 180,E1 -1157.71,E2 -1157.71} C_VEL
LIN {X 0,Y 594.301,Z 527.53,A -85,B 0,C 180,E1 -1157.926,E2 -1157.926} C_VEL
LIN {X 0,Y 594.68,Z 533.227,A -85,B 0,C 180,E1 -1158.042,E2 -1158.042} C_VEL
LIN {X 0,Y 594.639,Z 546.494,A -85,B 0,C 180,E1 -1158.366,E2 -1158.366} C_VEL
LIN {X 0,Y 594.587,Z 558.362,A -85,B 0,C 180,E1 -1158.79,E2 -1158.79} C_VEL
LIN {X 0,Y 594.511,Z 570.208,A -85,B 0,C 180,E1 -1159.356,E2 -1159.356} C_VEL
LIN {X 0,Y 594.462,Z 581.476,A -85,B 0,C 180,E1 -1160.043,E2 -1160.043} C_VEL
LIN {X 0,Y 594.406,Z 591.646,A -85,B 0,C 180,E1 -1160.815,E2 -1160.815} C_VEL
LIN {X 0,Y 594.372,Z 600.787,A -85,B 0,C 180,E1 -1161.672,E2 -1161.672} C_VEL
LIN {X 0,Y 594.316,Z 609.691,A -85,B 0,C 180,E1 -1162.697,E2 -1162.697} C_VEL
LIN {X 0,Y 594.281,Z 616.168,A -85,B 0,C 180,E1 -1163.615,E2 -1163.615} C_VEL
LIN {X 0,Y 594.289,Z 621.68,A -85,B 0,C 180,E1 -1164.571,E2 -1164.571} C_VEL
LIN {X 0,Y 594.27,Z 626.371,A -85,B 0,C 180,E1 -1165.591,E2 -1165.591} C_VEL
LIN {X 0,Y 594.267,Z 629.956,A -85,B 0,C 180,E1 -1166.61,E2 -1166.61} C_VEL
LIN {X 0,Y 594.226,Z 631.809,A -85,B 0,C 180,E1 -1167.288,E2 -1167.288} C_VEL
LIN {X 0,Y 594.24,Z 633.202,A -85,B 0,C 180,E1 -1167.967,E2 -1167.967} C_VEL
LIN {X 0,Y 594.239,Z 634.784,A -85,B 0,C 180,E1 -1169.322,E2 -1169.322} C_VEL
LIN {X 0,Y 594.236,Z 635,A -85,B 0,C 180,E1 -1170,E2 -1170} C_VEL
LIN {X 0,Y 594.247,Z 634.185,A -85,B 0,C 180,E1 -1171.355,E2 -1171.355} C_VEL
LIN {X 0,Y 594.24,Z 633.202,A -85,B 0,C 180,E1 -1172.033,E2 -1172.033} C_VEL
LIN {X 0,Y 594.226,Z 631.809,A -85,B 0,C 180,E1 -1172.712,E2 -1172.712} C_VEL
LIN {X 0,Y 594.288,Z 628.896,A -85,B 0,C 180,E1 -1173.729,E2 -1173.729} C_VEL
LIN {X 0,Y 594.242,Z 624.95,A -85,B 0,C 180,E1 -1174.749,E2 -1174.749} C_VEL
LIN {X 0,Y 594.304,Z 618.877,A -85,B 0,C 180,E1 -1175.939,E2 -1175.939} C_VEL
LIN {X 0,Y 594.308,Z 612.236,A -85,B 0,C 180,E1 -1176.962,E2 -1176.962} C_VEL
LIN {X 0,Y 594.359,Z 603.989,A -85,B 0,C 180,E1 -1177.986,E2 -1177.986} C_VEL
LIN {X 0,Y 594.382,Z 595.536,A -85,B 0,C 180,E1 -1178.842,E2 -1178.842} C_VEL
LIN {X 0,Y 594.431,Z 585.092,A -85,B 0,C 180,E1 -1179.699,E2 -1179.699} C_VEL
LIN {X 0,Y 594.482,Z 574.757,A -85,B 0,C 180,E1 -1180.386,E2 -1180.386} C_VEL
LIN {X 0,Y 594.534,Z 563.746,A -85,B 0,C 180,E1 -1180.972,E2 -1180.972} C_VEL
LIN {X 0,Y 594.598,Z 551.716,A -85,B 0,C 180,E1 -1181.464,E2 -1181.464} C_VEL
LIN {X 0,Y 594.655,Z 538.349,A -85,B 0,C 180,E1 -1181.85,E2 -1181.85} C_VEL
LIN {X 0,Y 594.469,Z 528.858,A -85,B 0,C 180,E1 -1182.038,E2 -1182.038} C_VEL
LIN {X 0,Y 594.301,Z 527.53,A -85,B 0,C 180,E1 -1182.074,E2 -1182.074} C_VEL
LIN {X 0,Y 594.317,Z 517.435,A -85,B 0,C 180,E1 -1184.729,E2 -1184.729} C_VEL
LIN {X 0,Y 594.334,Z 506.844,A -85,B 0,C 180,E1 -1187.55,E2 -1187.55} C_VEL
LIN {X 0,Y 594.381,Z 496.253,A -85,B 0,C 180,E1 -1190.415,E2 -1190.415} C_VEL
LIN {X 0,Y 594.437,Z 485.661,A -85,B 0,C 180,E1 -1193.333,E2 -1193.333} C_VEL
LIN {X 0,Y 594.484,Z 476.034,A -85,B 0,C 180,E1 -1196.042,E2 -1196.042} C_VEL
LIN {X 0,Y 594.507,Z 467.143,A -85,B 0,C 180,E1 -1198.601,E2 -1198.601} C_VEL
LIN {X 0,Y 594.55,Z 459.081,A -85,B 0,C 180,E1 -1200.944,E2 -1200.944} C_VEL
LIN {X 0,Y 594.587,Z 451.111,A -85,B 0,C 180,E1 -1203.341,E2 -1203.341} C_VEL
LIN {X 0,Y 594.641,Z 444.866,A -85,B 0,C 180,E1 -1205.389,E2 -1205.389} C_VEL
LIN {X 0,Y 594.36,Z 442.452,A -85,B 0,C 180,E1 -1206.333,E2 -1206.333} C_VEL
LIN {X 0,Y 594.39,Z 442.45,A -85,B 0,C 180,E1 -1208.805,E2 -1208.805} C_VEL
LIN {X 0,Y 594.384,Z 442.447,A -85,B 0,C 180,E1 -1211.848,E2 -1211.848} C_VEL
LIN {X 0,Y 594.367,Z 442.451,A -85,B 0,C 180,E1 -1214.809,E2 -1214.809} C_VEL
LIN {X 0,Y 594.373,Z 442.45,A -85,B 0,C 180,E1 -1217.625,E2 -1217.625} C_VEL
LIN {X 0,Y 594.394,Z 442.446,A -85,B 0,C 180,E1 -1220.321,E2 -1220.321} C_VEL
LIN {X 0,Y 594.386,Z 442.447,A -85,B 0,C 180,E1 -1222.913,E2 -1222.913} C_VEL
LIN {X 0,Y 594.315,Z 442.459,A -85,B 0,C 180,E1 -1224.682,E2 -1224.682} C_VEL
LIN {X 0,Y 594.308,Z 443.971,A -85,B 0,C 180,E1 -1226.234,E2 -1226.234} C_VEL
LIN {X 0,Y 594.326,Z 446.686,A -85,B 0,C 180,E1 -1228.647,E2 -1228.647} C_VEL
LIN {X 0,Y 594.258,Z 449.223,A -85,B 0,C 180,E1 -1231.065,E2 -1231.065} C_VEL
LIN {X 0,Y 594.296,Z 452.962,A -85,B 0,C 180,E1 -1234.052,E2 -1234.052} C_VEL
LIN {X 0,Y 594.243,Z 455.844,A -85,B 0,C 180,E1 -1236.29,E2 -1236.29} C_VEL
LIN {X 0,Y 594.296,Z 459.687,A -85,B 0,C 180,E1 -1239.221,E2 -1239.221} C_VEL
LIN {X 0,Y 594.209,Z 463.531,A -85,B 0,C 180,E1 -1242.091,E2 -1242.091} C_VEL
LIN {X 0,Y 594.248,Z 466.413,A -85,B 0,C 180,E1 -1244.216,E2 -1244.216} C_VEL
LIN {X 0,Y 594.239,Z 470.257,A -85,B 0,C 180,E1 -1247.014,E2 -1247.014} C_VEL
LIN {X 0,Y 594.258,Z 471.668,A -85,B 0,C 180,E1 -1248.034,E2 -1248.034} C_VEL
LIN {X 0,Y 594.645,Z 476.451,A -85,B 0,C 180,E1 -1248.15,E2 -1248.15} C_VEL
LIN {X 0,Y 594.592,Z 489.103,A -85,B 0,C 180,E1 -1248.494,E2 -1248.494} C_VEL
LIN {X 0,Y 594.533,Z 501.521,A -85,B 0,C 180,E1 -1248.972,E2 -1248.972} C_VEL
LIN {X 0,Y 594.502,Z 512.526,A -85,B 0,C 180,E1 -1249.528,E2 -1249.528} C_VEL
LIN {X 0,Y 594.447,Z 523.318,A -85,B 0,C 180,E1 -1250.215,E2 -1250.215} C_VEL
LIN {X 0,Y 594.404,Z 533.092,A -85,B 0,C 180,E1 -1250.987,E2 -1250.987} C_VEL
LIN {X 0,Y 594.366,Z 541.987,A -85,B 0,C 180,E1 -1251.843,E2 -1251.843} C_VEL
LIN {X 0,Y 594.345,Z 550.672,A -85,B 0,C 180,E1 -1252.868,E2 -1252.868} C_VEL
LIN {X 0,Y 594.29,Z 557.601,A -85,B 0,C 180,E1 -1253.89,E2 -1253.89} C_VEL
LIN {X 0,Y 594.254,Z 563.152,A -85,B 0,C 180,E1 -1254.911,E2 -1254.911} C_VEL
LIN {X 0,Y 594.262,Z 567.514,A -85,B 0,C 180,E1 -1255.931,E2 -1255.931} C_VEL
LIN {X 0,Y 594.268,Z 569.817,A -85,B 0,C 180,E1 -1256.61,E2 -1256.61} C_VEL
LIN {X 0,Y 594.225,Z 571.695,A -85,B 0,C 180,E1 -1257.289,E2 -1257.289} C_VEL
LIN {X 0,Y 594.24,Z 573.128,A -85,B 0,C 180,E1 -1257.967,E2 -1257.967} C_VEL
LIN {X 0,Y 594.24,Z 574.753,A -85,B 0,C 180,E1 -1259.323,E2 -1259.323} C_VEL
LIN {X 0,Y 594.236,Z 574.996,A -85,B 0,C 180,E1 -1260,E2 -1260} C_VEL
LIN {X 0,Y 594.24,Z 574.815,A -85,B 0,C 180,E1 -1260.678,E2 -1260.678} C_VEL
LIN {X 0,Y 594.239,Z 573.275,A -85,B 0,C 180,E1 -1262.033,E2 -1262.033} C_VEL
LIN {X 0,Y 594.226,Z 571.914,A -85,B 0,C 180,E1 -1262.712,E2 -1262.712} C_VEL
LIN {X 0,Y 594.289,Z 569.037,A -85,B 0,C 180,E1 -1263.729,E2 -1263.729} C_VEL
LIN {X 0,Y 594.242,Z 565.138,A -85,B 0,C 180,E1 -1264.749,E2 -1264.749} C_VEL
LIN {X 0,Y 594.299,Z 560.106,A -85,B 0,C 180,E1 -1265.769,E2 -1265.769} C_VEL
LIN {X 0,Y 594.316,Z 553.786,A -85,B 0,C 180,E1 -1266.792,E2 -1266.792} C_VEL
LIN {X 0,Y 594.346,Z 545.868,A -85,B 0,C 180,E1 -1267.816,E2 -1267.816} C_VEL
LIN {X 0,Y 594.381,Z 536.021,A -85,B 0,C 180,E1 -1268.842,E2 -1268.842} C_VEL
LIN {X 0,Y 594.427,Z 525.699,A -85,B 0,C 180,E1 -1269.7,E2 -1269.7} C_VEL
LIN {X 0,Y 594.502,Z 514.075,A -85,B 0,C 180,E1 -1270.472,E2 -1270.472} C_VEL
LIN {X 0,Y 594.56,Z 502.29,A -85,B 0,C 180,E1 -1271.084,E2 -1271.084} C_VEL
LIN {X 0,Y 594.598,Z 489.223,A -85,B 0,C 180,E1 -1271.592,E2 -1271.592} C_VEL
LIN {X 0,Y 594.64,Z 481.725,A -85,B 0,C 180,E1 -1271.814,E2 -1271.814} C_VEL
LIN {X 0,Y 594.335,Z 478.385,A -85,B 0,C 180,E1 -1271.968,E2 -1271.968} C_VEL
LIN {X 0,Y 593.466,Z 475.678,A -85,B 0,C 180,E1 -1272.207,E2 -1272.207} C_VEL
LIN {X 0,Y 591.622,Z 472.703,A -85,B 0,C 180,E1 -1272.661,E2 -1272.661} C_VEL
LIN {X 0,Y 589.572,Z 470.804,A -85,B 0,C 180,E1 -1273.202,E2 -1273.202} C_VEL
LIN {X 0,Y 587.484,Z 469.246,A -85,B 0,C 180,E1 -1273.992,E2 -1273.992} C_VEL
LIN {X 0,Y 587.148,Z 468.669,A -85,B 0,C 180,E1 -1274.403,E2 -1274.403} C_VEL
LIN {X 0,Y 587.147,Z 465.503,A -85,B 0,C 180,E1 -1276.748,E2 -1276.748} C_VEL
LIN {X 0,Y 587.138,Z 461.728,A -85,B 0,C 180,E1 -1279.582,E2 -1279.582} C_VEL
LIN {X 0,Y 587.142,Z 458.844,A -85,B 0,C 180,E1 -1281.782,E2 -1281.782} C_VEL
LIN {X 0,Y 587.178,Z 454.998,A -85,B 0,C 180,E1 -1284.767,E2 -1284.767} C_VEL
LIN {X 0,Y 587.197,Z 451.354,A -85,B 0,C 180,E1 -1287.664,E2 -1287.664} C_VEL
LIN {X 0,Y 587.232,Z 448.126,A -85,B 0,C 180,E1 -1290.492,E2 -1290.492} C_VEL
LIN {X 0,Y 587.22,Z 444.654,A -85,B 0,C 180,E1 -1293.404,E2 -1293.404} C_VEL
LIN {X 0,Y 587.234,Z 443.555,A -85,B 0,C 180,E1 -1294.331,E2 -1294.331} C_VEL
LIN {X 0,Y 587.353,Z 443.323,A -85,B 0,C 180,E1 -1296.747,E2 -1296.747} C_VEL
LIN {X 0,Y 587.334,Z 443.321,A -85,B 0,C 180,E1 -1299.361,E2 -1299.361} C_VEL
LIN {X 0,Y 587.34,Z 443.328,A -85,B 0,C 180,E1 -1302.108,E2 -1302.108} C_VEL
LIN {X 0,Y 587.322,Z 443.324,A -85,B 0,C 180,E1 -1305.089,E2 -1305.089} C_VEL
LIN {X 0,Y 587.326,Z 443.323,A -85,B 0,C 180,E1 -1307.925,E2 -1307.925} C_VEL
LIN {X 0,Y 587.338,Z 443.328,A -85,B 0,C 180,E1 -1310.64,E2 -1310.64} C_VEL
LIN {X 0,Y 587.352,Z 443.318,A -85,B 0,C 180,E1 -1313.293,E2 -1313.293} C_VEL
LIN {X 0,Y 587.372,Z 443.323,A -85,B 0,C 180,E1 -1315.781,E2 -1315.781} C_VEL
LIN {X 0,Y 587.348,Z 443.32,A -85,B 0,C 180,E1 -1318.231,E2 -1318.231} C_VEL
LIN {X 0,Y 587.355,Z 443.324,A -85,B 0,C 180,E1 -1320.867,E2 -1320.867} C_VEL
LIN {X 0,Y 587.366,Z 443.318,A -85,B 0,C 180,E1 -1323.819,E2 -1323.819} C_VEL
LIN {X 0,Y 587.333,Z 443.326,A -85,B 0,C 180,E1 -1325.993,E2 -1325.993} C_VEL
LIN {X 0,Y 587.324,Z 443.325,A -85,B 0,C 180,E1 -1328.226,E2 -1328.226} C_VEL
LIN {X 0,Y 587.355,Z 443.324,A -85,B 0,C 180,E1 -1331.151,E2 -1331.151} C_VEL
LIN {X 0,Y 587.322,Z 443.323,A -85,B 0,C 180,E1 -1334.025,E2 -1334.025} C_VEL
LIN {X 0,Y 587.365,Z 443.321,A -85,B 0,C 180,E1 -1336.154,E2 -1336.154} C_VEL
LIN {X 0,Y 587.344,Z 443.319,A -85,B 0,C 180,E1 -1338.962,E2 -1338.962} C_VEL
LIN {X 0,Y 587.369,Z 443.322,A -85,B 0,C 180,E1 -1341.745,E2 -1341.745} C_VEL
LIN {X 0,Y 587.359,Z 443.319,A -85,B 0,C 180,E1 -1344.507,E2 -1344.507} C_VEL
LIN {X 0,Y 587.372,Z 443.318,A -85,B 0,C 180,E1 -1347.257,E2 -1347.257} C_VEL
LIN {X 0,Y 587.389,Z 443.319,A -85,B 0,C 180,E1 -1350,E2 -1350} C_VEL
LIN {X 0,Y 587.372,Z 443.316,A -85,B 0,C 180,E1 -1352.743,E2 -1352.743} C_VEL
LIN {X 0,Y 587.365,Z 443.323,A -85,B 0,C 180,E1 -1355.493,E2 -1355.493} C_VEL
LIN {X 0,Y 587.349,Z 443.321,A -85,B 0,C 180,E1 -1358.256,E2 -1358.256} C_VEL
LIN {X 0,Y 587.355,Z 443.319,A -85,B 0,C 180,E1 -1361.134,E2 -1361.134} C_VEL
LIN {X 0,Y 587.372,Z 443.319,A -85,B 0,C 180,E1 -1364.26,E2 -1364.26} C_VEL
LIN {X 0,Y 587.351,Z 443.326,A -85,B 0,C 180,E1 -1367.406,E2 -1367.406} C_VEL
LIN {X 0,Y 587.332,Z 443.323,A -85,B 0,C 180,E1 -1370.305,E2 -1370.305} C_VEL
LIN {X 0,Y 587.32,Z 443.323,A -85,B 0,C 180,E1 -1373.259,E2 -1373.259} C_VEL
LIN {X 0,Y 587.336,Z 443.323,A -85,B 0,C 180,E1 -1375.517,E2 -1375.517} C_VEL
LIN {X 0,Y 587.345,Z 443.325,A -85,B 0,C 180,E1 -1377.818,E2 -1377.818} C_VEL
LIN {X 0,Y 587.341,Z 443.321,A -85,B 0,C 180,E1 -1380.51,E2 -1380.51} C_VEL
LIN {X 0,Y 587.338,Z 443.321,A -85,B 0,C 180,E1 -1383.397,E2 -1383.397} C_VEL
LIN {X 0,Y 587.304,Z 443.328,A -85,B 0,C 180,E1 -1385.899,E2 -1385.899} C_VEL
LIN {X 0,Y 587.327,Z 443.323,A -85,B 0,C 180,E1 -1388.48,E2 -1388.48} C_VEL
LIN {X 0,Y 587.34,Z 443.325,A -85,B 0,C 180,E1 -1391.157,E2 -1391.157} C_VEL
LIN {X 0,Y 587.317,Z 443.324,A -85,B 0,C 180,E1 -1394.112,E2 -1394.112} C_VEL
LIN {X 0,Y 587.326,Z 443.324,A -85,B 0,C 180,E1 -1396.994,E2 -1396.994} C_VEL
LIN {X 0,Y 587.316,Z 443.328,A -85,B 0,C 180,E1 -1399.745,E2 -1399.745} C_VEL
LIN {X 0,Y 587.348,Z 443.319,A -85,B 0,C 180,E1 -1402.392,E2 -1402.392} C_VEL
LIN {X 0,Y 587.305,Z 443.33,A -85,B 0,C 180,E1 -1404.942,E2 -1404.942} C_VEL
LIN {X 0,Y 587.244,Z 443.339,A -85,B 0,C 180,E1 -1405.772,E2 -1405.772} C_VEL
LIN {X 0,Y 587.197,Z 445.133,A -85,B 0,C 180,E1 -1407.412,E2 -1407.412} C_VEL
LIN {X 0,Y 587.192,Z 448.121,A -85,B 0,C 180,E1 -1409.821,E2 -1409.821} C_VEL
LIN {X 0,Y 587.197,Z 451.242,A -85,B 0,C 180,E1 -1412.336,E2 -1412.336} C_VEL
LIN {X 0,Y 587.178,Z 454.884,A -85,B 0,C 180,E1 -1415.233,E2 -1415.233} C_VEL
LIN {X 0,Y 587.143,Z 458.727,A -85,B 0,C 180,E1 -1418.218,E2 -1418.218} C_VEL
LIN {X 0,Y 587.154,Z 462.399,A -85,B 0,C 180,E1 -1421.015,E2 -1421.015} C_VEL
LIN {X 0,Y 587.155,Z 466.413,A -85,B 0,C 180,E1 -1424.02,E2 -1424.02} C_VEL
LIN {X 0,Y 587.14,Z 470.257,A -85,B 0,C 180,E1 -1426.854,E2 -1426.854} C_VEL
LIN {X 0,Y 587.156,Z 471.668,A -85,B 0,C 180,E1 -1427.887,E2 -1427.887} C_VEL
LIN {X 0,Y 587.701,Z 477.294,A -85,B 0,C 180,E1 -1428.029,E2 -1428.029} C_VEL
LIN {X 0,Y 587.655,Z 489.27,A -85,B 0,C 180,E1 -1428.362,E2 -1428.362} C_VEL
LIN {X 0,Y 587.571,Z 501.324,A -85,B 0,C 180,E1 -1428.83,E2 -1428.83} C_VEL
LIN {X 0,Y 587.503,Z 514.007,A -85,B 0,C 180,E1 -1429.489,E2 -1429.489} C_VEL
LIN {X 0,Y 587.424,Z 524.459,A -85,B 0,C 180,E1 -1430.184,E2 -1430.184} C_VEL
LIN {X 0,Y 587.357,Z 533.068,A -85,B 0,C 180,E1 -1430.877,E2 -1430.877} C_VEL
LIN {X 0,Y 587.302,Z 541.976,A -85,B 0,C 180,E1 -1431.744,E2 -1431.744} C_VEL
LIN {X 0,Y 587.274,Z 550.675,A -85,B 0,C 180,E1 -1432.781,E2 -1432.781} C_VEL
LIN {X 0,Y 587.214,Z 557.601,A -85,B 0,C 180,E1 -1433.816,E2 -1433.816} C_VEL
LIN {X 0,Y 587.167,Z 563.146,A -85,B 0,C 180,E1 -1434.849,E2 -1434.849} C_VEL
LIN {X 0,Y 587.182,Z 567.498,A -85,B 0,C 180,E1 -1435.882,E2 -1435.882} C_VEL
LIN {X 0,Y 587.194,Z 569.824,A -85,B 0,C 180,E1 -1436.569,E2 -1436.569} C_VEL
LIN {X 0,Y 587.132,Z 571.685,A -85,B 0,C 180,E1 -1437.255,E2 -1437.255} C_VEL
LIN {X 0,Y 587.139,Z 573.112,A -85,B 0,C 180,E1 -1437.942,E2 -1437.942} C_VEL
LIN {X 0,Y 587.146,Z 574.135,A -85,B 0,C 180,E1 -1438.628,E2 -1438.628} C_VEL
LIN {X 0,Y 587.141,Z 574.753,A -85,B 0,C 180,E1 -1439.314,E2 -1439.314} C_VEL
LIN {X 0,Y 587.14,Z 574.811,A -85,B 0,C 180,E1 -1440.686,E2 -1440.686} C_VEL
LIN {X 0,Y 587.148,Z 574.24,A -85,B 0,C 180,E1 -1441.372,E2 -1441.372} C_VEL
LIN {X 0,Y 587.133,Z 571.91,A -85,B 0,C 180,E1 -1442.744,E2 -1442.744} C_VEL
LIN {X 0,Y 587.213,Z 569.039,A -85,B 0,C 180,E1 -1443.774,E2 -1443.774} C_VEL
LIN {X 0,Y 587.147,Z 565.138,A -85,B 0,C 180,E1 -1444.806,E2 -1444.806} C_VEL
LIN {X 0,Y 587.229,Z 560.092,A -85,B 0,C 180,E1 -1445.839,E2 -1445.839} C_VEL
LIN {X 0,Y 587.229,Z 553.758,A -85,B 0,C 180,E1 -1446.874,E2 -1446.874} C_VEL
LIN {X 0,Y 587.288,Z 545.875,A -85,B 0,C 180,E1 -1447.91,E2 -1447.91} C_VEL
LIN {X 0,Y 587.33,Z 536.007,A -85,B 0,C 180,E1 -1448.949,E2 -1448.949} C_VEL
LIN {X 0,Y 587.419,Z 526.819,A -85,B 0,C 180,E1 -1449.729,E2 -1449.729} C_VEL
LIN {X 0,Y 587.482,Z 516.883,A -85,B 0,C 180,E1 -1450.424,E2 -1450.424} C_VEL
LIN {X 0,Y 587.547,Z 505.03,A -85,B 0,C 180,E1 -1451.086,E2 -1451.086} C_VEL
LIN {X 0,Y 587.621,Z 491.925,A -85,B 0,C 180,E1 -1451.638,E2 -1451.638} C_VEL
LIN {X 0,Y 587.69,Z 479.247,A -85,B 0,C 180,E1 -1452.014,E2 -1452.014} C_VEL
LIN {X 0,Y 587.486,Z 473.911,A -85,B 0,C 180,E1 -1452.139,E2 -1452.139} C_VEL
LIN {X 0,Y 587.155,Z 471.672,A -85,B 0,C 180,E1 -1452.201,E2 -1452.201} C_VEL
LIN {X 0,Y 587.131,Z 468.458,A -85,B 0,C 180,E1 -1454.559,E2 -1454.559} C_VEL
LIN {X 0,Y 587.146,Z 465.503,A -85,B 0,C 180,E1 -1456.747,E2 -1456.747} C_VEL
LIN {X 0,Y 587.135,Z 461.729,A -85,B 0,C 180,E1 -1459.582,E2 -1459.582} C_VEL
LIN {X 0,Y 587.143,Z 458.844,A -85,B 0,C 180,E1 -1461.781,E2 -1461.781} C_VEL
LIN {X 0,Y 587.179,Z 454.999,A -85,B 0,C 180,E1 -1464.766,E2 -1464.766} C_VEL
LIN {X 0,Y 587.166,Z 452.114,A -85,B 0,C 180,E1 -1467.054,E2 -1467.054} C_VEL
LIN {X 0,Y 587.168,Z 449.113,A -85,B 0,C 180,E1 -1469.389,E2 -1469.389} C_VEL
LIN {X 0,Y 587.175,Z 445.696,A -85,B 0,C 180,E1 -1471.808,E2 -1471.808} C_VEL
LIN {X 0,Y 587.153,Z 443.35,A -85,B 0,C 180,E1 -1473.408,E2 -1473.408} C_VEL
LIN {X 0,Y 587.296,Z 443.331,A -85,B 0,C 180,E1 -1475.9,E2 -1475.9} C_VEL
LIN {X 0,Y 587.325,Z 443.327,A -85,B 0,C 180,E1 -1478.48,E2 -1478.48} C_VEL
LIN {X 0,Y 587.34,Z 443.325,A -85,B 0,C 180,E1 -1481.157,E2 -1481.157} C_VEL
LIN {X 0,Y 587.338,Z 443.324,A -85,B 0,C 180,E1 -1484.114,E2 -1484.114} C_VEL
LIN {X 0,Y 587.315,Z 443.329,A -85,B 0,C 180,E1 -1486.993,E2 -1486.993} C_VEL
LIN {X 0,Y 587.321,Z 443.33,A -85,B 0,C 180,E1 -1489.746,E2 -1489.746} C_VEL
LIN {X 0,Y 587.346,Z 443.327,A -85,B 0,C 180,E1 -1492.392,E2 -1492.392} C_VEL
LIN {X 0,Y 587.348,Z 443.361,A -85,B 0,C 180,E1 -1493.679,E2 -1493.679} C_VEL
LIN {X 0,Y 587.687,Z 447.249,A -85,B 0,C 180,E1 -1494.969,E2 -1494.969} C_VEL
LIN {X 0,Y 587.642,Z 456.319,A -85,B 0,C 180,E1 -1497.823,E2 -1497.823} C_VEL
LIN {X 0,Y 587.563,Z 465.774,A -85,B 0,C 180,E1 -1500.632,E2 -1500.632} C_VEL
LIN {X 0,Y 587.507,Z 475.07,A -85,B 0,C 180,E1 -1503.347,E2 -1503.347} C_VEL
LIN {X 0,Y 587.414,Z 484.338,A -85,B 0,C 180,E1 -1505.997,E2 -1505.997} C_VEL
LIN {X 0,Y 587.357,Z 493.606,A -85,B 0,C 180,E1 -1508.596,E2 -1508.596} C_VEL
LIN {X 0,Y 587.323,Z 504.196,A -85,B 0,C 180,E1 -1511.512,E2 -1511.512} C_VEL
LIN {X 0,Y 587.261,Z 514.787,A -85,B 0,C 180,E1 -1514.379,E2 -1514.379} C_VEL
LIN {X 0,Y 587.24,Z 524.055,A -85,B 0,C 180,E1 -1516.857,E2 -1516.857} C_VEL
LIN {X 0,Y 587.215,Z 527.571,A -85,B 0,C 180,E1 -1517.789,E2 -1517.789} C_VEL
LIN {X 0,Y 587.736,Z 533.227,A -85,B 0,C 180,E1 -1517.899,E2 -1517.899} C_VEL
LIN {X 0,Y 587.681,Z 546.495,A -85,B 0,C 180,E1 -1518.226,E2 -1518.226} C_VEL
LIN {X 0,Y 587.622,Z 558.273,A -85,B 0,C 180,E1 -1518.651,E2 -1518.651} C_VEL
LIN {X 0,Y 587.528,Z 570.209,A -85,B 0,C 180,E1 -1519.228,E2 -1519.228} C_VEL
LIN {X 0,Y 587.457,Z 581.477,A -85,B 0,C 180,E1 -1519.923,E2 -1519.923} C_VEL
LIN {X 0,Y 587.384,Z 591.646,A -85,B 0,C 180,E1 -1520.704,E2 -1520.704} C_VEL
LIN {X 0,Y 587.34,Z 600.787,A -85,B 0,C 180,E1 -1521.571,E2 -1521.571} C_VEL
LIN {X 0,Y 587.259,Z 609.69,A -85,B 0,C 180,E1 -1522.608,E2 -1522.608} C_VEL
LIN {X 0,Y 587.195,Z 616.745,A -85,B 0,C 180,E1 -1523.627,E2 -1523.627} C_VEL
LIN {X 0,Y 587.211,Z 621.68,A -85,B 0,C 180,E1 -1524.506,E2 -1524.506} C_VEL
LIN {X 0,Y 587.188,Z 626.371,A -85,B 0,C 180,E1 -1525.538,E2 -1525.538} C_VEL
LIN {X 0,Y 587.194,Z 629.956,A -85,B 0,C 180,E1 -1526.569,E2 -1526.569} C_VEL
LIN {X 0,Y 587.132,Z 631.809,A -85,B 0,C 180,E1 -1527.256,E2 -1527.256} C_VEL
LIN {X 0,Y 587.139,Z 633.201,A -85,B 0,C 180,E1 -1527.942,E2 -1527.942} C_VEL
LIN {X 0,Y 587.14,Z 634.784,A -85,B 0,C 180,E1 -1529.314,E2 -1529.314} C_VEL
LIN {X 0,Y 587.137,Z 635,A -85,B 0,C 180,E1 -1530,E2 -1530} C_VEL
LIN {X 0,Y 587.147,Z 634.185,A -85,B 0,C 180,E1 -1531.372,E2 -1531.372} C_VEL
LIN {X 0,Y 587.139,Z 633.201,A -85,B 0,C 180,E1 -1532.058,E2 -1532.058} C_VEL
LIN {X 0,Y 587.132,Z 631.81,A -85,B 0,C 180,E1 -1532.744,E2 -1532.744} C_VEL
LIN {X 0,Y 587.212,Z 628.896,A -85,B 0,C 180,E1 -1533.774,E2 -1533.774} C_VEL
LIN {X 0,Y 587.147,Z 624.949,A -85,B 0,C 180,E1 -1534.806,E2 -1534.806} C_VEL
LIN {X 0,Y 587.217,Z 618.877,A -85,B 0,C 180,E1 -1536.011,E2 -1536.011} C_VEL
LIN {X 0,Y 587.245,Z 612.236,A -85,B 0,C 180,E1 -1537.046,E2 -1537.046} C_VEL
LIN {X 0,Y 587.299,Z 603.989,A -85,B 0,C 180,E1 -1538.083,E2 -1538.083} C_VEL
LIN {X 0,Y 587.343,Z 595.537,A -85,B 0,C 180,E1 -1538.949,E2 -1538.949} C_VEL
LIN {X 0,Y 587.417,Z 585.094,A -85,B 0,C 180,E1 -1539.816,E2 -1539.816} C_VEL
LIN {X 0,Y 587.501,Z 574.758,A -85,B 0,C 180,E1 -1540.511,E2 -1540.511} C_VEL
LIN {X 0,Y 587.557,Z 562.853,A -85,B 0,C 180,E1 -1541.147,E2 -1541.147} C_VEL
LIN {X 0,Y 587.637,Z 550.617,A -85,B 0,C 180,E1 -1541.638,E2 -1541.638} C_VEL
LIN {X 0,Y 587.722,Z 537.434,A -85,B 0,C 180,E1 -1542.014,E2 -1542.014} C_VEL
LIN {X 0,Y 587.505,Z 529.608,A -85,B 0,C 180,E1 -1542.172,E2 -1542.172} C_VEL
LIN {X 0,Y 587.214,Z 527.53,A -85,B 0,C 180,E1 -1542.221,E2 -1542.221} C_VEL
LIN {X 0,Y 587.269,Z 517.435,A -85,B 0,C 180,E1 -1544.91,E2 -1544.91} C_VEL
LIN {X 0,Y 587.302,Z 506.844,A -85,B 0,C 180,E1 -1547.767,E2 -1547.767} C_VEL
LIN {X 0,Y 587.375,Z 496.253,A -85,B 0,C 180,E1 -1550.669,E2 -1550.669} C_VEL
LIN {X 0,Y 587.432,Z 485.661,A -85,B 0,C 180,E1 -1553.628,E2 -1553.628} C_VEL
LIN {X 0,Y 587.486,Z 476.394,A -85,B 0,C 180,E1 -1556.272,E2 -1556.272} C_VEL
LIN {X 0,Y 587.517,Z 467.457,A -85,B 0,C 180,E1 -1558.877,E2 -1558.877} C_VEL
LIN {X 0,Y 587.546,Z 458.92,A -85,B 0,C 180,E1 -1561.355,E2 -1561.355} C_VEL
LIN {X 0,Y 587.633,Z 451.079,A -85,B 0,C 180,E1 -1563.789,E2 -1563.789} C_VEL
LIN {X 0,Y 587.65,Z 445.046,A -85,B 0,C 180,E1 -1565.875,E2 -1565.875} C_VEL
LIN {X 0,Y 587.352,Z 443.326,A -85,B 0,C 180,E1 -1566.645,E2 -1566.645} C_VEL
LIN {X 0,Y 587.349,Z 443.324,A -85,B 0,C 180,E1 -1569.359,E2 -1569.359} C_VEL
LIN {X 0,Y 587.338,Z 443.325,A -85,B 0,C 180,E1 -1572.108,E2 -1572.108} C_VEL
LIN {X 0,Y 587.32,Z 443.33,A -85,B 0,C 180,E1 -1575.089,E2 -1575.089} C_VEL
LIN {X 0,Y 587.356,Z 443.323,A -85,B 0,C 180,E1 -1577.928,E2 -1577.928} C_VEL
LIN {X 0,Y 587.338,Z 443.328,A -85,B 0,C 180,E1 -1581.058,E2 -1581.058} C_VEL
LIN {X 0,Y 587.351,Z 443.325,A -85,B 0,C 180,E1 -1583.293,E2 -1583.293} C_VEL
LIN {X 0,Y 587.26,Z 443.338,A -85,B 0,C 180,E1 -1584.94,E2 -1584.94} C_VEL
LIN {X 0,Y 587.261,Z 446.026,A -85,B 0,C 180,E1 -1587.416,E2 -1587.416} C_VEL
LIN {X 0,Y 587.237,Z 448.721,A -85,B 0,C 180,E1 -1589.824,E2 -1589.824} C_VEL
LIN {X 0,Y 587.196,Z 451.259,A -85,B 0,C 180,E1 -1592.337,E2 -1592.337} C_VEL
LIN {X 0,Y 587.175,Z 453.924,A -85,B 0,C 180,E1 -1594.476,E2 -1594.476} C_VEL
LIN {X 0,Y 587.149,Z 457.37,A -85,B 0,C 180,E1 -1597.172,E2 -1597.172} C_VEL
LIN {X 0,Y 587.168,Z 460.649,A -85,B 0,C 180,E1 -1599.689,E2 -1599.689} C_VEL
LIN {X 0,Y 587.13,Z 464.492,A -85,B 0,C 180,E1 -1602.587,E2 -1602.587} C_VEL
LIN {X 0,Y 587.148,Z 468.336,A -85,B 0,C 180,E1 -1605.442,E2 -1605.442} C_VEL
LIN {X 0,Y 587.135,Z 471.669,A -85,B 0,C 180,E1 -1607.887,E2 -1607.887} C_VEL
LIN {X 0,Y 587.697,Z 477.389,A -85,B 0,C 180,E1 -1608.03,E2 -1608.03} C_VEL
LIN {X 0,Y 587.622,Z 490.656,A -85,B 0,C 180,E1 -1608.408,E2 -1608.408} C_VEL
LIN {X 0,Y 587.565,Z 502.014,A -85,B 0,C 180,E1 -1608.861,E2 -1608.861} C_VEL
LIN {X 0,Y 587.502,Z 514.024,A -85,B 0,C 180,E1 -1609.489,E2 -1609.489} C_VEL
LIN {X 0,Y 587.399,Z 525.656,A -85,B 0,C 180,E1 -1610.27,E2 -1610.27} C_VEL
LIN {X 0,Y 587.344,Z 535.038,A -85,B 0,C 180,E1 -1611.051,E2 -1611.051} C_VEL
LIN {X 0,Y 587.3,Z 543.601,A -85,B 0,C 180,E1 -1611.917,E2 -1611.917} C_VEL
LIN {X 0,Y 587.262,Z 551.915,A -85,B 0,C 180,E1 -1612.954,E2 -1612.954} C_VEL
LIN {X 0,Y 587.218,Z 558.615,A -85,B 0,C 180,E1 -1613.989,E2 -1613.989} C_VEL
LIN {X 0,Y 587.146,Z 564.759,A -85,B 0,C 180,E1 -1615.194,E2 -1615.194} C_VEL
LIN {X 0,Y 587.213,Z 568.748,A -85,B 0,C 180,E1 -1616.226,E2 -1616.226} C_VEL
LIN {X 0,Y 587.132,Z 571.697,A -85,B 0,C 180,E1 -1617.256,E2 -1617.256} C_VEL
LIN {X 0,Y 587.139,Z 573.128,A -85,B 0,C 180,E1 -1617.942,E2 -1617.942} C_VEL
LIN {X 0,Y 587.14,Z 574.754,A -85,B 0,C 180,E1 -1619.314,E2 -1619.314} C_VEL
LIN {X 0,Y 587.137,Z 574.996,A -85,B 0,C 180,E1 -1620,E2 -1620} C_VEL
LIN {X 0,Y 587.14,Z 574.815,A -85,B 0,C 180,E1 -1620.686,E2 -1620.686} C_VEL
LIN {X 0,Y 587.138,Z 573.274,A -85,B 0,C 180,E1 -1622.058,E2 -1622.058} C_VEL
LIN {X 0,Y 587.133,Z 571.913,A -85,B 0,C 180,E1 -1622.745,E2 -1622.745} C_VEL
LIN {X 0,Y 587.213,Z 569.035,A -85,B 0,C 180,E1 -1623.774,E2 -1623.774} C_VEL
LIN {X 0,Y 587.147,Z 565.135,A -85,B 0,C 180,E1 -1624.807,E2 -1624.807} C_VEL
LIN {X 0,Y 587.229,Z 560.103,A -85,B 0,C 180,E1 -1625.839,E2 -1625.839} C_VEL
LIN {X 0,Y 587.23,Z 553.782,A -85,B 0,C 180,E1 -1626.874,E2 -1626.874} C_VEL
LIN {X 0,Y 587.288,Z 545.863,A -85,B 0,C 180,E1 -1627.91,E2 -1627.91} C_VEL
LIN {X 0,Y 587.343,Z 536.015,A -85,B 0,C 180,E1 -1628.949,E2 -1628.949} C_VEL
LIN {X 0,Y 587.411,Z 525.693,A -85,B 0,C 180,E1 -1629.817,E2 -1629.817} C_VEL
LIN {X 0,Y 587.505,Z 514.064,A -85,B 0,C 180,E1 -1630.599,E2 -1630.599} C_VEL
LIN {X 0,Y 587.591,Z 503.112,A -85,B 0,C 180,E1 -1631.18,E2 -1631.18} C_VEL
LIN {X 0,Y 587.624,Z 490.445,A -85,B 0,C 180,E1 -1631.69,E2 -1631.69} C_VEL
LIN {X 0,Y 587.702,Z 477.479,A -85,B 0,C 180,E1 -1632.058,E2 -1632.058} C_VEL
LIN {X 0,Y 587.372,Z 473.277,A -85,B 0,C 180,E1 -1632.153,E2 -1632.153} C_VEL
LIN {X 0,Y 587.14,Z 471.672,A -85,B 0,C 180,E1 -1632.201,E2 -1632.201} C_VEL
LIN {X 0,Y 587.148,Z 468.669,A -85,B 0,C 180,E1 -1634.403,E2 -1634.403} C_VEL
LIN {X 0,Y 586.479,Z 467.922,A -85,B 0,C 180,E1 -1634.971,E2 -1634.971} C_VEL
LIN {X 0,Y 583.6,Z 466.785,A -85,B 0,C 180,E1 -1635.893,E2 -1635.893} C_VEL
LIN {X 0,Y 581.167,Z 465.887,A -85,B 0,C 180,E1 -1636.636,E2 -1636.636} C_VEL
LIN {X 0,Y 580.124,Z 465.168,A -85,B 0,C 180,E1 -1637.209,E2 -1637.209} C_VEL
LIN {X 0,Y 580.04,Z 464.916,A -85,B 0,C 180,E1 -1637.402,E2 -1637.402} C_VEL
LIN {X 0,Y 580.066,Z 461.727,A -85,B 0,C 180,E1 -1639.831,E2 -1639.831} C_VEL
LIN {X 0,Y 580.046,Z 458.843,A -85,B 0,C 180,E1 -1642.062,E2 -1642.062} C_VEL
LIN {X 0,Y 580.096,Z 455.511,A -85,B 0,C 180,E1 -1644.681,E2 -1644.681} C_VEL
LIN {X 0,Y 580.119,Z 452.24,A -85,B 0,C 180,E1 -1647.411,E2 -1647.411} C_VEL
LIN {X 0,Y 580.137,Z 449.542,A -85,B 0,C 180,E1 -1649.782,E2 -1649.782} C_VEL
LIN {X 0,Y 580.139,Z 446.642,A -85,B 0,C 180,E1 -1652.211,E2 -1652.211} C_VEL
LIN {X 0,Y 580.17,Z 444.693,A -85,B 0,C 180,E1 -1653.865,E2 -1653.865} C_VEL
LIN {X 0,Y 580.196,Z 444.218,A -85,B 0,C 180,E1 -1654.703,E2 -1654.703} C_VEL
LIN {X 0,Y 580.303,Z 444.2,A -85,B 0,C 180,E1 -1657.269,E2 -1657.269} C_VEL
LIN {X 0,Y 580.293,Z 444.204,A -85,B 0,C 180,E1 -1660.27,E2 -1660.27} C_VEL
LIN {X 0,Y 580.287,Z 444.2,A -85,B 0,C 180,E1 -1662.706,E2 -1662.706} C_VEL
LIN {X 0,Y 580.267,Z 444.209,A -85,B 0,C 180,E1 -1665.61,E2 -1665.61} C_VEL
LIN {X 0,Y 580.284,Z 444.2,A -85,B 0,C 180,E1 -1668.231,E2 -1668.231} C_VEL
LIN {X 0,Y 580.284,Z 444.203,A -85,B 0,C 180,E1 -1670.965,E2 -1670.965} C_VEL
LIN {X 0,Y 580.274,Z 444.201,A -85,B 0,C 180,E1 -1673.597,E2 -1673.597} C_VEL
LIN {X 0,Y 580.324,Z 444.198,A -85,B 0,C 180,E1 -1676.146,E2 -1676.146} C_VEL
LIN {X 0,Y 580.282,Z 444.2,A -85,B 0,C 180,E1 -1678.615,E2 -1678.615} C_VEL
LIN {X 0,Y 580.297,Z 444.205,A -85,B 0,C 180,E1 -1681.024,E2 -1681.024} C_VEL
LIN {X 0,Y 580.297,Z 444.198,A -85,B 0,C 180,E1 -1683.666,E2 -1683.666} C_VEL
LIN {X 0,Y 580.303,Z 444.198,A -85,B 0,C 180,E1 -1685.684,E2 -1685.684} C_VEL
LIN {X 0,Y 580.291,Z 444.198,A -85,B 0,C 180,E1 -1688.695,E2 -1688.695} C_VEL
LIN {X 0,Y 580.304,Z 444.199,A -85,B 0,C 180,E1 -1690.913,E2 -1690.913} C_VEL
LIN {X 0,Y 580.272,Z 444.201,A -85,B 0,C 180,E1 -1693.825,E2 -1693.825} C_VEL
LIN {X 0,Y 580.332,Z 444.195,A -85,B 0,C 180,E1 -1695.983,E2 -1695.983} C_VEL
LIN {X 0,Y 580.312,Z 444.196,A -85,B 0,C 180,E1 -1698.827,E2 -1698.827} C_VEL
LIN {X 0,Y 580.332,Z 444.201,A -85,B 0,C 180,E1 -1701.644,E2 -1701.644} C_VEL
LIN {X 0,Y 580.325,Z 444.195,A -85,B 0,C 180,E1 -1704.44,E2 -1704.44} C_VEL
LIN {X 0,Y 580.339,Z 444.194,A -85,B 0,C 180,E1 -1707.223,E2 -1707.223} C_VEL
LIN {X 0,Y 580.359,Z 444.195,A -85,B 0,C 180,E1 -1710,E2 -1710} C_VEL
LIN {X 0,Y 580.339,Z 444.192,A -85,B 0,C 180,E1 -1712.777,E2 -1712.777} C_VEL
LIN {X 0,Y 580.329,Z 444.198,A -85,B 0,C 180,E1 -1715.56,E2 -1715.56} C_VEL
LIN {X 0,Y 580.317,Z 444.198,A -85,B 0,C 180,E1 -1718.356,E2 -1718.356} C_VEL
LIN {X 0,Y 580.307,Z 444.197,A -85,B 0,C 180,E1 -1721.191,E2 -1721.191} C_VEL
LIN {X 0,Y 580.332,Z 444.199,A -85,B 0,C 180,E1 -1724.017,E2 -1724.017} C_VEL
LIN {X 0,Y 580.319,Z 444.197,A -85,B 0,C 180,E1 -1726.914,E2 -1726.914} C_VEL
LIN {X 0,Y 580.293,Z 444.198,A -85,B 0,C 180,E1 -1729.823,E2 -1729.823} C_VEL
LIN {X 0,Y 580.277,Z 444.202,A -85,B 0,C 180,E1 -1732.053,E2 -1732.053} C_VEL
LIN {X 0,Y 580.311,Z 444.196,A -85,B 0,C 180,E1 -1735.08,E2 -1735.08} C_VEL
LIN {X 0,Y 580.3,Z 444.198,A -85,B 0,C 180,E1 -1738.186,E2 -1738.186} C_VEL
LIN {X 0,Y 580.291,Z 444.201,A -85,B 0,C 180,E1 -1740.695,E2 -1740.695} C_VEL
LIN {X 0,Y 580.307,Z 444.198,A -85,B 0,C 180,E1 -1743.316,E2 -1743.316} C_VEL
LIN {X 0,Y 580.268,Z 444.203,A -85,B 0,C 180,E1 -1745.758,E2 -1745.758} C_VEL
LIN {X 0,Y 580.29,Z 444.203,A -85,B 0,C 180,E1 -1748.146,E2 -1748.146} C_VEL
LIN {X 0,Y 580.302,Z 444.198,A -85,B 0,C 180,E1 -1750.843,E2 -1750.843} C_VEL
LIN {X 0,Y 580.278,Z 444.201,A -85,B 0,C 180,E1 -1753.658,E2 -1753.658} C_VEL
LIN {X 0,Y 580.29,Z 444.205,A -85,B 0,C 180,E1 -1756.608,E2 -1756.608} C_VEL
LIN {X 0,Y 580.302,Z 444.197,A -85,B 0,C 180,E1 -1759.156,E2 -1759.156} C_VEL
LIN {X 0,Y 580.292,Z 444.202,A -85,B 0,C 180,E1 -1761.927,E2 -1761.927} C_VEL
LIN {X 0,Y 580.254,Z 444.203,A -85,B 0,C 180,E1 -1764.452,E2 -1764.452} C_VEL
LIN {X 0,Y 580.156,Z 444.221,A -85,B 0,C 180,E1 -1766.134,E2 -1766.134} C_VEL
LIN {X 0,Y 580.123,Z 447.096,A -85,B 0,C 180,E1 -1768.605,E2 -1768.605} C_VEL
LIN {X 0,Y 580.099,Z 450.15,A -85,B 0,C 180,E1 -1771.013,E2 -1771.013} C_VEL
LIN {X 0,Y 580.118,Z 453.376,A -85,B 0,C 180,E1 -1773.701,E2 -1773.701} C_VEL
LIN {X 0,Y 580.067,Z 456.806,A -85,B 0,C 180,E1 -1776.433,E2 -1776.433} C_VEL
LIN {X 0,Y 580.087,Z 460.649,A -85,B 0,C 180,E1 -1779.43,E2 -1779.43} C_VEL
LIN {X 0,Y 580.042,Z 464.493,A -85,B 0,C 180,E1 -1782.367,E2 -1782.367} C_VEL
LIN {X 0,Y 580.057,Z 467.375,A -85,B 0,C 180,E1 -1784.54,E2 -1784.54} C_VEL
LIN {X 0,Y 580.073,Z 471.219,A -85,B 0,C 180,E1 -1787.403,E2 -1787.403} C_VEL
LIN {X 0,Y 580.075,Z 471.669,A -85,B 0,C 180,E1 -1787.737,E2 -1787.737} C_VEL
LIN {X 0,Y 580.774,Z 477.292,A -85,B 0,C 180,E1 -1787.885,E2 -1787.885} C_VEL
LIN {X 0,Y 580.697,Z 489.106,A -85,B 0,C 180,E1 -1788.215,E2 -1788.215} C_VEL
LIN {X 0,Y 580.596,Z 500.68,A -85,B 0,C 180,E1 -1788.665,E2 -1788.665} C_VEL
LIN {X 0,Y 580.536,Z 512.55,A -85,B 0,C 180,E1 -1789.273,E2 -1789.273} C_VEL
LIN {X 0,Y 580.439,Z 523.298,A -85,B 0,C 180,E1 -1789.976,E2 -1789.976} C_VEL
LIN {X 0,Y 580.333,Z 533.066,A -85,B 0,C 180,E1 -1790.766,E2 -1790.766} C_VEL
LIN {X 0,Y 580.264,Z 541.977,A -85,B 0,C 180,E1 -1791.643,E2 -1791.643} C_VEL
LIN {X 0,Y 580.206,Z 550.679,A -85,B 0,C 180,E1 -1792.693,E2 -1792.693} C_VEL
LIN {X 0,Y 580.137,Z 557.604,A -85,B 0,C 180,E1 -1793.74,E2 -1793.74} C_VEL
LIN {X 0,Y 580.085,Z 563.147,A -85,B 0,C 180,E1 -1794.786,E2 -1794.786} C_VEL
LIN {X 0,Y 580.105,Z 567.495,A -85,B 0,C 180,E1 -1795.831,E2 -1795.831} C_VEL
LIN {X 0,Y 580.123,Z 569.828,A -85,B 0,C 180,E1 -1796.527,E2 -1796.527} C_VEL
LIN {X 0,Y 580.043,Z 571.684,A -85,B 0,C 180,E1 -1797.222,E2 -1797.222} C_VEL
LIN {X 0,Y 580.046,Z 574.137,A -85,B 0,C 180,E1 -1798.611,E2 -1798.611} C_VEL
LIN {X 0,Y 580.041,Z 574.754,A -85,B 0,C 180,E1 -1799.306,E2 -1799.306} C_VEL
LIN {X 0,Y 580.04,Z 574.81,A -85,B 0,C 180,E1 -1800.694,E2 -1800.694} C_VEL
LIN {X 0,Y 580.048,Z 574.241,A -85,B 0,C 180,E1 -1801.388,E2 -1801.388} C_VEL
LIN {X 0,Y 580.044,Z 571.906,A -85,B 0,C 180,E1 -1802.778,E2 -1802.778} C_VEL
LIN {X 0,Y 580.11,Z 569.034,A -85,B 0,C 180,E1 -1803.82,E2 -1803.82} C_VEL
LIN {X 0,Y 580.053,Z 565.13,A -85,B 0,C 180,E1 -1804.865,E2 -1804.865} C_VEL
LIN {X 0,Y 580.162,Z 560.082,A -85,B 0,C 180,E1 -1805.91,E2 -1805.91} C_VEL
LIN {X 0,Y 580.157,Z 553.746,A -85,B 0,C 180,E1 -1806.958,E2 -1806.958} C_VEL
LIN {X 0,Y 580.241,Z 545.873,A -85,B 0,C 180,E1 -1808.007,E2 -1808.007} C_VEL
LIN {X 0,Y 580.299,Z 535.993,A -85,B 0,C 180,E1 -1809.058,E2 -1809.058} C_VEL
LIN {X 0,Y 580.382,Z 526.802,A -85,B 0,C 180,E1 -1809.848,E2 -1809.848} C_VEL
LIN {X 0,Y 580.492,Z 516.861,A -85,B 0,C 180,E1 -1810.551,E2 -1810.551} C_VEL
LIN {X 0,Y 580.57,Z 506.073,A -85,B 0,C 180,E1 -1811.168,E2 -1811.168} C_VEL
LIN {X 0,Y 580.66,Z 493.02,A -85,B 0,C 180,E1 -1811.741,E2 -1811.741} C_VEL
LIN {X 0,Y 580.749,Z 480.106,A -85,B 0,C 180,E1 -1812.138,E2 -1812.138} C_VEL
LIN {X 0,Y 580.544,Z 474.846,A -85,B 0,C 180,E1 -1812.268,E2 -1812.268} C_VEL
LIN {X 0,Y 580.09,Z 471.671,A -85,B 0,C 180,E1 -1812.352,E2 -1812.352} C_VEL
LIN {X 0,Y 580.047,Z 468.457,A -85,B 0,C 180,E1 -1814.74,E2 -1814.74} C_VEL
LIN {X 0,Y 580.066,Z 465.573,A -85,B 0,C 180,E1 -1816.905,E2 -1816.905} C_VEL
LIN {X 0,Y 580.064,Z 461.728,A -85,B 0,C 180,E1 -1819.831,E2 -1819.831} C_VEL
LIN {X 0,Y 580.046,Z 458.844,A -85,B 0,C 180,E1 -1822.062,E2 -1822.062} C_VEL
LIN {X 0,Y 580.097,Z 455.511,A -85,B 0,C 180,E1 -1824.681,E2 -1824.681} C_VEL
LIN {X 0,Y 580.089,Z 452.066,A -85,B 0,C 180,E1 -1827.412,E2 -1827.412} C_VEL
LIN {X 0,Y 580.072,Z 448.988,A -85,B 0,C 180,E1 -1829.785,E2 -1829.785} C_VEL
LIN {X 0,Y 580.066,Z 445.439,A -85,B 0,C 180,E1 -1832.215,E2 -1832.215} C_VEL
LIN {X 0,Y 580.078,Z 444.232,A -85,B 0,C 180,E1 -1833.039,E2 -1833.039} C_VEL
LIN {X 0,Y 580.26,Z 444.207,A -85,B 0,C 180,E1 -1834.698,E2 -1834.698} C_VEL
LIN {X 0,Y 580.302,Z 444.202,A -85,B 0,C 180,E1 -1837.268,E2 -1837.268} C_VEL
LIN {X 0,Y 580.294,Z 444.202,A -85,B 0,C 180,E1 -1840.27,E2 -1840.27} C_VEL
LIN {X 0,Y 580.285,Z 444.203,A -85,B 0,C 180,E1 -1842.706,E2 -1842.706} C_VEL
LIN {X 0,Y 580.273,Z 444.205,A -85,B 0,C 180,E1 -1845.609,E2 -1845.609} C_VEL
LIN {X 0,Y 580.283,Z 444.205,A -85,B 0,C 180,E1 -1848.231,E2 -1848.231} C_VEL
LIN {X 0,Y 580.293,Z 444.206,A -85,B 0,C 180,E1 -1850.966,E2 -1850.966} C_VEL
LIN {X 0,Y 580.33,Z 444.394,A -85,B 0,C 180,E1 -1853.506,E2 -1853.506} C_VEL
LIN {X 0,Y 580.753,Z 448.571,A -85,B 0,C 180,E1 -1854.913,E2 -1854.913} C_VEL
LIN {X 0,Y 580.672,Z 457.69,A -85,B 0,C 180,E1 -1857.822,E2 -1857.822} C_VEL
LIN {X 0,Y 580.564,Z 467.055,A -85,B 0,C 180,E1 -1860.645,E2 -1860.645} C_VEL
LIN {X 0,Y 580.484,Z 477.219,A -85,B 0,C 180,E1 -1863.628,E2 -1863.628} C_VEL
LIN {X 0,Y 580.418,Z 485.661,A -85,B 0,C 180,E1 -1866.069,E2 -1866.069} C_VEL
LIN {X 0,Y 580.323,Z 495.405,A -85,B 0,C 180,E1 -1868.83,E2 -1868.83} C_VEL
LIN {X 0,Y 580.251,Z 505.52,A -85,B 0,C 180,E1 -1871.644,E2 -1871.644} C_VEL
LIN {X 0,Y 580.2,Z 516.111,A -85,B 0,C 180,E1 -1874.545,E2 -1874.545} C_VEL
LIN {X 0,Y 580.166,Z 526.703,A -85,B 0,C 180,E1 -1877.406,E2 -1877.406} C_VEL
LIN {X 0,Y 580.146,Z 527.53,A -85,B 0,C 180,E1 -1877.627,E2 -1877.627} C_VEL
LIN {X 0,Y 580.813,Z 533.227,A -85,B 0,C 180,E1 -1877.753,E2 -1877.753} C_VEL
LIN {X 0,Y 580.737,Z 546.495,A -85,B 0,C 180,E1 -1878.083,E2 -1878.083} C_VEL
LIN {X 0,Y 580.659,Z 558.524,A -85,B 0,C 180,E1 -1878.525,E2 -1878.525} C_VEL
LIN {X 0,Y 580.531,Z 570.211,A -85,B 0,C 180,E1 -1879.096,E2 -1879.096} C_VEL
LIN {X 0,Y 580.447,Z 581.478,A -85,B 0,C 180,E1 -1879.8,E2 -1879.8} C_VEL
LIN {X 0,Y 580.352,Z 591.646,A -85,B 0,C 180,E1 -1880.591,E2 -1880.591} C_VEL
LIN {X 0,Y 580.279,Z 600.787,A -85,B 0,C 180,E1 -1881.468,E2 -1881.468} C_VEL
LIN {X 0,Y 580.199,Z 609.69,A -85,B 0,C 180,E1 -1882.518,E2 -1882.518} C_VEL
LIN {X 0,Y 580.12,Z 616.465,A -85,B 0,C 180,E1 -1883.505,E2 -1883.505} C_VEL
LIN {X 0,Y 580.139,Z 621.68,A -85,B 0,C 180,E1 -1884.438,E2 -1884.438} C_VEL
LIN {X 0,Y 580.108,Z 626.372,A -85,B 0,C 180,E1 -1885.483,E2 -1885.483} C_VEL
LIN {X 0,Y 580.123,Z 629.957,A -85,B 0,C 180,E1 -1886.527,E2 -1886.527} C_VEL
LIN {X 0,Y 580.043,Z 631.808,A -85,B 0,C 180,E1 -1887.222,E2 -1887.222} C_VEL
LIN {X 0,Y 580.038,Z 633.2,A -85,B 0,C 180,E1 -1887.917,E2 -1887.917} C_VEL
LIN {X 0,Y 580.04,Z 634.784,A -85,B 0,C 180,E1 -1889.306,E2 -1889.306} C_VEL
LIN {X 0,Y 580.037,Z 635,A -85,B 0,C 180,E1 -1890,E2 -1890} C_VEL
LIN {X 0,Y 580.047,Z 634.185,A -85,B 0,C 180,E1 -1891.389,E2 -1891.389} C_VEL
LIN {X 0,Y 580.038,Z 633.201,A -85,B 0,C 180,E1 -1892.083,E2 -1892.083} C_VEL
LIN {X 0,Y 580.043,Z 631.81,A -85,B 0,C 180,E1 -1892.778,E2 -1892.778} C_VEL
LIN {X 0,Y 580.109,Z 628.896,A -85,B 0,C 180,E1 -1893.821,E2 -1893.821} C_VEL
LIN {X 0,Y 580.054,Z 624.949,A -85,B 0,C 180,E1 -1894.865,E2 -1894.865} C_VEL
LIN {X 0,Y 580.139,Z 618.877,A -85,B 0,C 180,E1 -1896.085,E2 -1896.085} C_VEL
LIN {X 0,Y 580.184,Z 612.237,A -85,B 0,C 180,E1 -1897.132,E2 -1897.132} C_VEL
LIN {X 0,Y 580.25,Z 603.99,A -85,B 0,C 180,E1 -1898.182,E2 -1898.182} C_VEL
LIN {X 0,Y 580.308,Z 595.537,A -85,B 0,C 180,E1 -1899.058,E2 -1899.058} C_VEL
LIN {X 0,Y 580.417,Z 585.095,A -85,B 0,C 180,E1 -1899.936,E2 -1899.936} C_VEL
LIN {X 0,Y 580.506,Z 574.756,A -85,B 0,C 180,E1 -1900.639,E2 -1900.639} C_VEL
LIN {X 0,Y 580.584,Z 563.371,A -85,B 0,C 180,E1 -1901.258,E2 -1901.258} C_VEL
LIN {X 0,Y 580.675,Z 551.765,A -85,B 0,C 180,E1 -1901.741,E2 -1901.741} C_VEL
LIN {X 0,Y 580.776,Z 538.347,A -85,B 0,C 180,E1 -1902.137,E2 -1902.137} C_VEL
LIN {X 0,Y 580.578,Z 530.328,A -85,B 0,C 180,E1 -1902.308,E2 -1902.308} C_VEL
LIN {X 0,Y 580.146,Z 527.53,A -85,B 0,C 180,E1 -1902.373,E2 -1902.373} C_VEL
LIN {X 0,Y 580.226,Z 517.435,A -85,B 0,C 180,E1 -1905.095,E2 -1905.095} C_VEL
LIN {X 0,Y 580.253,Z 506.844,A -85,B 0,C 180,E1 -1907.99,E2 -1907.99} C_VEL
LIN {X 0,Y 580.344,Z 496.491,A -85,B 0,C 180,E1 -1910.865,E2 -1910.865} C_VEL
LIN {X 0,Y 580.404,Z 486.985,A -85,B 0,C 180,E1 -1913.553,E2 -1913.553} C_VEL
LIN {X 0,Y 580.455,Z 479.042,A -85,B 0,C 180,E1 -1915.841,E2 -1915.841} C_VEL
LIN {X 0,Y 580.521,Z 470.966,A -85,B 0,C 180,E1 -1918.174,E2 -1918.174} C_VEL
LIN {X 0,Y 580.575,Z 462.215,A -85,B 0,C 180,E1 -1920.742,E2 -1920.742} C_VEL
LIN {X 0,Y 580.623,Z 454.859,A -85,B 0,C 180,E1 -1923.004,E2 -1923.004} C_VEL
LIN {X 0,Y 580.734,Z 447.539,A -85,B 0,C 180,E1 -1925.513,E2 -1925.513} C_VEL
LIN {X 0,Y 580.301,Z 444.203,A -85,B 0,C 180,E1 -1926.934,E2 -1926.934} C_VEL
LIN {X 0,Y 580.299,Z 444.204,A -85,B 0,C 180,E1 -1929.933,E2 -1929.933} C_VEL
LIN {X 0,Y 580.279,Z 444.207,A -85,B 0,C 180,E1 -1932.706,E2 -1932.706} C_VEL
LIN {X 0,Y 580.278,Z 444.204,A -85,B 0,C 180,E1 -1935.609,E2 -1935.609} C_VEL
LIN {X 0,Y 580.317,Z 444.2,A -85,B 0,C 180,E1 -1938.234,E2 -1938.234} C_VEL
LIN {X 0,Y 580.293,Z 444.205,A -85,B 0,C 180,E1 -1940.966,E2 -1940.966} C_VEL
LIN {X 0,Y 580.267,Z 444.209,A -85,B 0,C 180,E1 -1943.596,E2 -1943.596} C_VEL
LIN {X 0,Y 580.21,Z 444.484,A -85,B 0,C 180,E1 -1945.298,E2 -1945.298} C_VEL
LIN {X 0,Y 580.219,Z 447.384,A -85,B 0,C 180,E1 -1947.983,E2 -1947.983} C_VEL
LIN {X 0,Y 580.166,Z 450.656,A -85,B 0,C 180,E1 -1951.017,E2 -1951.017} C_VEL
LIN {X 0,Y 580.129,Z 453.389,A -85,B 0,C 180,E1 -1953.699,E2 -1953.699} C_VEL
LIN {X 0,Y 580.069,Z 456.807,A -85,B 0,C 180,E1 -1956.433,E2 -1956.433} C_VEL
LIN {X 0,Y 580.086,Z 460.65,A -85,B 0,C 180,E1 -1959.43,E2 -1959.43} C_VEL
LIN {X 0,Y 580.041,Z 464.493,A -85,B 0,C 180,E1 -1962.368,E2 -1962.368} C_VEL
LIN {X 0,Y 580.058,Z 467.376,A -85,B 0,C 180,E1 -1964.541,E2 -1964.541} C_VEL
LIN {X 0,Y 580.059,Z 470.258,A -85,B 0,C 180,E1 -1966.691,E2 -1966.691} C_VEL
LIN {X 0,Y 580.061,Z 471.67,A -85,B 0,C 180,E1 -1967.737,E2 -1967.737} C_VEL
LIN {X 0,Y 580.762,Z 477.411,A -85,B 0,C 180,E1 -1967.885,E2 -1967.885} C_VEL
LIN {X 0,Y 580.695,Z 490.454,A -85,B 0,C 180,E1 -1968.26,E2 -1968.26} C_VEL
LIN {X 0,Y 580.58,Z 502.488,A -85,B 0,C 180,E1 -1968.746,E2 -1968.746} C_VEL
LIN {X 0,Y 580.517,Z 514.032,A -85,B 0,C 180,E1 -1969.361,E2 -1969.361} C_VEL
LIN {X 0,Y 580.389,Z 525.665,A -85,B 0,C 180,E1 -1970.152,E2 -1970.152} C_VEL
LIN {X 0,Y 580.308,Z 535.044,A -85,B 0,C 180,E1 -1970.942,E2 -1970.942} C_VEL
LIN {X 0,Y 580.251,Z 543.606,A -85,B 0,C 180,E1 -1971.818,E2 -1971.818} C_VEL
LIN {X 0,Y 580.205,Z 551.919,A -85,B 0,C 180,E1 -1972.868,E2 -1972.868} C_VEL
LIN {X 0,Y 580.14,Z 558.618,A -85,B 0,C 180,E1 -1973.915,E2 -1973.915} C_VEL
LIN {X 0,Y 580.053,Z 564.761,A -85,B 0,C 180,E1 -1975.135,E2 -1975.135} C_VEL
LIN {X 0,Y 580.11,Z 568.75,A -85,B 0,C 180,E1 -1976.18,E2 -1976.18} C_VEL
LIN {X 0,Y 580.043,Z 571.698,A -85,B 0,C 180,E1 -1977.222,E2 -1977.222} C_VEL
LIN {X 0,Y 580.038,Z 573.128,A -85,B 0,C 180,E1 -1977.917,E2 -1977.917} C_VEL
LIN {X 0,Y 580.041,Z 574.755,A -85,B 0,C 180,E1 -1979.306,E2 -1979.306} C_VEL
LIN {X 0,Y 580.038,Z 574.996,A -85,B 0,C 180,E1 -1980,E2 -1980} C_VEL
LIN {X 0,Y 580.04,Z 574.815,A -85,B 0,C 180,E1 -1980.694,E2 -1980.694} C_VEL
LIN {X 0,Y 580.037,Z 573.272,A -85,B 0,C 180,E1 -1982.083,E2 -1982.083} C_VEL
LIN {X 0,Y 580.044,Z 571.911,A -85,B 0,C 180,E1 -1982.778,E2 -1982.778} C_VEL
LIN {X 0,Y 580.11,Z 569.033,A -85,B 0,C 180,E1 -1983.821,E2 -1983.821} C_VEL
LIN {X 0,Y 580.054,Z 565.133,A -85,B 0,C 180,E1 -1984.865,E2 -1984.865} C_VEL
LIN {X 0,Y 580.161,Z 560.1,A -85,B 0,C 180,E1 -1985.91,E2 -1985.91} C_VEL
LIN {X 0,Y 580.158,Z 553.778,A -85,B 0,C 180,E1 -1986.958,E2 -1986.958} C_VEL
LIN {X 0,Y 580.241,Z 545.858,A -85,B 0,C 180,E1 -1988.007,E2 -1988.007} C_VEL
LIN {X 0,Y 580.308,Z 536.009,A -85,B 0,C 180,E1 -1989.059,E2 -1989.059} C_VEL
LIN {X 0,Y 580.41,Z 525.687,A -85,B 0,C 180,E1 -1989.936,E2 -1989.936} C_VEL
LIN {X 0,Y 580.503,Z 514.054,A -85,B 0,C 180,E1 -1990.728,E2 -1990.728} C_VEL
LIN {X 0,Y 580.631,Z 502.285,A -85,B 0,C 180,E1 -1991.353,E2 -1991.353} C_VEL
LIN {X 0,Y 580.688,Z 490.616,A -85,B 0,C 180,E1 -1991.825,E2 -1991.825} C_VEL
LIN {X 0,Y 580.77,Z 477.455,A -85,B 0,C 180,E1 -1992.204,E2 -1992.204} C_VEL
LIN {X 0,Y 580.079,Z 471.671,A -85,B 0,C 180,E1 -1992.352,E2 -1992.352} C_VEL
LIN {X 0,Y 580.058,Z 468.457,A -85,B 0,C 180,E1 -1994.74,E2 -1994.74} C_VEL
LIN {X 0,Y 580.04,Z 464.916,A -85,B 0,C 180,E1 -1997.402,E2 -1997.402} C_VEL
LIN {X 0,Y 579.373,Z 464.185,A -85,B 0,C 180,E1 -1997.978,E2 -1997.978} C_VEL
LIN {X 0,Y 576.511,Z 463.085,A -85,B 0,C 180,E1 -1998.913,E2 -1998.913} C_VEL
LIN {X 0,Y 574.092,Z 462.218,A -85,B 0,C 180,E1 -1999.665,E2 -1999.665} C_VEL
LIN {X 0,Y 573.057,Z 461.519,A -85,B 0,C 180,E1 -2000.245,E2 -2000.245} C_VEL
LIN {X 0,Y 572.974,Z 461.271,A -85,B 0,C 180,E1 -2000.442,E2 -2000.442} C_VEL
LIN {X 0,Y 572.991,Z 457.881,A -85,B 0,C 180,E1 -2003.11,E2 -2003.11} C_VEL
LIN {X 0,Y 572.995,Z 455.057,A -85,B 0,C 180,E1 -2005.423,E2 -2005.423} C_VEL
LIN {X 0,Y 573.068,Z 452.212,A -85,B 0,C 180,E1 -2007.994,E2 -2007.994} C_VEL
LIN {X 0,Y 573.061,Z 448.627,A -85,B 0,C 180,E1 -2011.004,E2 -2011.004} C_VEL
LIN {X 0,Y 573.077,Z 445.718,A -85,B 0,C 180,E1 -2013.495,E2 -2013.495} C_VEL
LIN {X 0,Y 573.117,Z 445.101,A -85,B 0,C 180,E1 -2014.339,E2 -2014.339} C_VEL
LIN {X 0,Y 573.256,Z 445.08,A -85,B 0,C 180,E1 -2017.166,E2 -2017.166} C_VEL
LIN {X 0,Y 573.242,Z 445.076,A -85,B 0,C 180,E1 -2019.608,E2 -2019.608} C_VEL
LIN {X 0,Y 573.249,Z 445.077,A -85,B 0,C 180,E1 -2022.642,E2 -2022.642} C_VEL
LIN {X 0,Y 573.228,Z 445.083,A -85,B 0,C 180,E1 -2025.325,E2 -2025.325} C_VEL
LIN {X 0,Y 573.244,Z 445.079,A -85,B 0,C 180,E1 -2027.6,E2 -2027.6} C_VEL
LIN {X 0,Y 573.25,Z 445.081,A -85,B 0,C 180,E1 -2030.568,E2 -2030.568} C_VEL
LIN {X 0,Y 573.257,Z 445.075,A -85,B 0,C 180,E1 -2033.078,E2 -2033.078} C_VEL
LIN {X 0,Y 573.277,Z 445.077,A -85,B 0,C 180,E1 -2035.672,E2 -2035.672} C_VEL
LIN {X 0,Y 573.247,Z 445.077,A -85,B 0,C 180,E1 -2038.185,E2 -2038.185} C_VEL
LIN {X 0,Y 573.27,Z 445.076,A -85,B 0,C 180,E1 -2040.634,E2 -2040.634} C_VEL
LIN {X 0,Y 573.243,Z 445.077,A -85,B 0,C 180,E1 -2043.508,E2 -2043.508} C_VEL
LIN {X 0,Y 573.232,Z 445.085,A -85,B 0,C 180,E1 -2046.134,E2 -2046.134} C_VEL
LIN {X 0,Y 573.257,Z 445.077,A -85,B 0,C 180,E1 -2049.174,E2 -2049.174} C_VEL
LIN {X 0,Y 573.228,Z 445.085,A -85,B 0,C 180,E1 -2051.411,E2 -2051.411} C_VEL
LIN {X 0,Y 573.247,Z 445.077,A -85,B 0,C 180,E1 -2053.622,E2 -2053.622} C_VEL
LIN {X 0,Y 573.28,Z 445.072,A -85,B 0,C 180,E1 -2055.807,E2 -2055.807} C_VEL
